  MoveL (T10079) to (119.5, 116.18, 12.1) mm, rotated rx 180 ry 0 rz -180 deg; joints [0, 0, 0, 0, 0, 0]
  Call Extruder -0.04075
  MoveL (T10080) to (119.58, 116.26, 12.1) mm, rotated rx 180 ry 0 rz -180 deg; joints [0, 0, 0, 0, 0, 0]
  Call Extruder -0.07305
  MoveL (T10081) to (119.79, 116.26, 12.1) mm, rotated rx 180 ry 0 rz -180 deg; joints [0, 0, 0, 0, 0, 0]
  Call Extruder -0.05902
  MoveL (T10082) to (119.9, 116.14, 12.1) mm, rotated rx 180 ry 0 rz -180 deg; joints [0, 0, 0, 0, 0, 0]
  Set speed (45.0 mm/s)
  Call Extruder -0.02
  MoveL (T10083) to (119.9, 116.14, 12.1) mm, rotated rx 180 ry 0 rz -180 deg; joints [0, 0, 0, 0, 0, 0]
  Set speed (150.0 mm/s)
  MoveL (T10084) to (119.9, 116.14, 14.1) mm, rotated rx 180 ry 0 rz -180 deg; joints [0, 0, 0, 0, 0, 0]
  MoveL (T10085) to (104.34, 103.54, 14.1) mm, rotated rx 180 ry 0 rz -180 deg; joints [0, 0, 0, 0, 0, 0]
  MoveL (T10086) to (104.34, 103.54, 12.3) mm, rotated rx 180 ry 0 rz -180 deg; joints [0, 0, 0, 0, 0, 0]
  Set speed (40.0 mm/s)
  Call Extruder 2.0
  MoveL (T10087) to (104.34, 103.54, 12.3) mm, rotated rx 180 ry 0 rz -180 deg; joints [0, 0, 0, 0, 0, 0]
  Set speed (26.4 mm/s)
  MoveL (T10088) to (104.34, 103.54, 12.3) mm, rotated rx 180 ry 0 rz -180 deg; joints [0, 0, 0, 0, 0, 0]
  Call Extruder 0.13732
  MoveL (T10089) to (108.85, 103.54, 12.3) mm, rotated rx 180 ry 0 rz -180 deg; joints [0, 0, 0, 0, 0, 0]
  Call Extruder 0.05783
  MoveL (T10090) to (108.85, 105.44, 12.3) mm, rotated rx 180 ry 0 rz -180 deg; joints [0, 0, 0, 0, 0, 0]
  Call Extruder 0.1948
  MoveL (T10091) to (115.24, 105.44, 12.3) mm, rotated rx 180 ry 0 rz -180 deg; joints [0, 0, 0, 0, 0, 0]
  Call Extruder 0.05783
  MoveL (T10092) to (115.24, 103.54, 12.3) mm, rotated rx 180 ry 0 rz -180 deg; joints [0, 0, 0, 0, 0, 0]
  Call Extruder 0.18953
  MoveL (T10093) to (121.46, 103.54, 12.3) mm, rotated rx 180 ry 0 rz -180 deg; joints [0, 0, 0, 0, 0, 0]
  Call Extruder 0.14944
  MoveL (T10094) to (121.46, 108.44, 12.3) mm, rotated rx 180 ry 0 rz -180 deg; joints [0, 0, 0, 0, 0, 0]
  Call Extruder 0.05883
  MoveL (T10095) to (119.53, 108.44, 12.3) mm, rotated rx 180 ry 0 rz -180 deg; joints [0, 0, 0, 0, 0, 0]
  Call Extruder 0.22006
  MoveL (T10096) to (119.53, 115.67, 12.3) mm, rotated rx 180 ry 0 rz -180 deg; joints [0, 0, 0, 0, 0, 0]
  Call Extruder 0.05893
  MoveL (T10097) to (121.46, 115.67, 12.3) mm, rotated rx 180 ry 0 rz -180 deg; joints [0, 0, 0, 0, 0, 0]
  Call Extruder 0.17636
  MoveL (T10098) to (121.46, 121.46, 12.3) mm, rotated rx 180 ry 0 rz -180 deg; joints [0, 0, 0, 0, 0, 0]
  Call Extruder 0.54596
  MoveL (T10099) to (103.54, 121.46, 12.3) mm, rotated rx 180 ry 0 rz -180 deg; joints [0, 0, 0, 0, 0, 0]
  Call Extruder 0.54596
  MoveL (T10100) to (103.54, 103.54, 12.3) mm, rotated rx 180 ry 0 rz -180 deg; joints [0, 0, 0, 0, 0, 0]
  Call Extruder 0.02254
  MoveL (T10101) to (104.28, 103.54, 12.3) mm, rotated rx 180 ry 0 rz -180 deg; joints [0, 0, 0, 0, 0, 0]
  Set speed (150.0 mm/s)
  MoveL (T10102) to (103.53, 103.13, 12.3) mm, rotated rx 180 ry 0 rz -180 deg; joints [0, 0, 0, 0, 0, 0]
  Set speed (26.4 mm/s)
  MoveL (T10103) to (103.53, 103.13, 12.3) mm, rotated rx 180 ry 0 rz -180 deg; joints [0, 0, 0, 0, 0, 0]
  Call Extruder 0.17431
  MoveL (T10104) to (109.25, 103.13, 12.3) mm, rotated rx 180 ry 0 rz -180 deg; joints [0, 0, 0, 0, 0, 0]
  Call Extruder 0.05783
  MoveL (T10105) to (109.25, 105.03, 12.3) mm, rotated rx 180 ry 0 rz -180 deg; joints [0, 0, 0, 0, 0, 0]
  Call Extruder 0.08214
  MoveL (T10106) to (111.95, 105.03, 12.3) mm, rotated rx 180 ry 0 rz -180 deg; joints [0, 0, 0, 0, 0, 0]
  Call Extruder 0.08784
  MoveL (T10107) to (114.83, 105.03, 12.3) mm, rotated rx 180 ry 0 rz -180 deg; joints [0, 0, 0, 0, 0, 0]
  Call Extruder 0.05783
  MoveL (T10108) to (114.83, 103.13, 12.3) mm, rotated rx 180 ry 0 rz -180 deg; joints [0, 0, 0, 0, 0, 0]
  Call Extruder 0.21434
  MoveL (T10109) to (121.87, 103.13, 12.3) mm, rotated rx 180 ry 0 rz -180 deg; joints [0, 0, 0, 0, 0, 0]
  Call Extruder 0.17423
  MoveL (T10110) to (121.87, 108.85, 12.3) mm, rotated rx 180 ry 0 rz -180 deg; joints [0, 0, 0, 0, 0, 0]
  Call Extruder 0.05884
  MoveL (T10111) to (119.94, 108.85, 12.3) mm, rotated rx 180 ry 0 rz -180 deg; joints [0, 0, 0, 0, 0, 0]
  Call Extruder 0.09005
  MoveL (T10112) to (119.94, 111.81, 12.3) mm, rotated rx 180 ry 0 rz -180 deg; joints [0, 0, 0, 0, 0, 0]
  Call Extruder 0.05887
  MoveL (T10113) to (121.87, 111.81, 12.3) mm, rotated rx 180 ry 0 rz -180 deg; joints [0, 0, 0, 0, 0, 0]
  Call Extruder 0.01564
  MoveL (T10114) to (121.87, 112.32, 12.3) mm, rotated rx 180 ry 0 rz -180 deg; joints [0, 0, 0, 0, 0, 0]
  Call Extruder 0.05888
  MoveL (T10115) to (119.94, 112.32, 12.3) mm, rotated rx 180 ry 0 rz -180 deg; joints [0, 0, 0, 0, 0, 0]
  Call Extruder 0.08969
  MoveL (T10116) to (119.93, 115.26, 12.3) mm, rotated rx 180 ry 0 rz -180 deg; joints [0, 0, 0, 0, 0, 0]
  Call Extruder 0.05892
  MoveL (T10117) to (121.87, 115.27, 12.3) mm, rotated rx 180 ry 0 rz -180 deg; joints [0, 0, 0, 0, 0, 0]
  Call Extruder 0.20115
  MoveL (T10118) to (121.87, 121.87, 12.3) mm, rotated rx 180 ry 0 rz -180 deg; joints [0, 0, 0, 0, 0, 0]
  Call Extruder 0.57077
  MoveL (T10119) to (103.13, 121.87, 12.3) mm, rotated rx 180 ry 0 rz -180 deg; joints [0, 0, 0, 0, 0, 0]
  Call Extruder 0.57077
  MoveL (T10120) to (103.13, 103.13, 12.3) mm, rotated rx 180 ry 0 rz -180 deg; joints [0, 0, 0, 0, 0, 0]
  Call Extruder 0.01036
  MoveL (T10121) to (103.47, 103.13, 12.3) mm, rotated rx 180 ry 0 rz -180 deg; joints [0, 0, 0, 0, 0, 0]
  Set speed (150.0 mm/s)
  MoveL (T10122) to (102.72, 102.81, 12.3) mm, rotated rx 180 ry 0 rz -180 deg; joints [0, 0, 0, 0, 0, 0]
  Set speed (25.0 mm/s)
  MoveL (T10123) to (102.72, 102.81, 12.3) mm, rotated rx 180 ry 0 rz -180 deg; joints [0, 0, 0, 0, 0, 0]
  Call Extruder 0.00259
  MoveL (T10124) to (102.72, 102.72, 12.3) mm, rotated rx 180 ry 0 rz -180 deg; joints [0, 0, 0, 0, 0, 0]
  Call Extruder 0.21131
  MoveL (T10125) to (109.66, 102.72, 12.3) mm, rotated rx 180 ry 0 rz -180 deg; joints [0, 0, 0, 0, 0, 0]
  Call Extruder 0.05783
  MoveL (T10126) to (109.66, 104.62, 12.3) mm, rotated rx 180 ry 0 rz -180 deg; joints [0, 0, 0, 0, 0, 0]
  Call Extruder 0.0643
  MoveL (T10127) to (111.77, 104.62, 12.3) mm, rotated rx 180 ry 0 rz -180 deg; joints [0, 0, 0, 0, 0, 0]
  Call Extruder 0.05783
  MoveL (T10128) to (111.77, 102.72, 12.3) mm, rotated rx 180 ry 0 rz -180 deg; joints [0, 0, 0, 0, 0, 0]
  Call Extruder 0.01777
  MoveL (T10129) to (112.36, 102.72, 12.3) mm, rotated rx 180 ry 0 rz -180 deg; joints [0, 0, 0, 0, 0, 0]
  Call Extruder 0.05783
  MoveL (T10130) to (112.36, 104.62, 12.3) mm, rotated rx 180 ry 0 rz -180 deg; joints [0, 0, 0, 0, 0, 0]
  Call Extruder 0.06304
  MoveL (T10131) to (114.43, 104.62, 12.3) mm, rotated rx 180 ry 0 rz -180 deg; joints [0, 0, 0, 0, 0, 0]
  Call Extruder 0.05783
  MoveL (T10132) to (114.42, 102.72, 12.3) mm, rotated rx 180 ry 0 rz -180 deg; joints [0, 0, 0, 0, 0, 0]
  Call Extruder 0.23915
  MoveL (T10133) to (122.28, 102.72, 12.3) mm, rotated rx 180 ry 0 rz -180 deg; joints [0, 0, 0, 0, 0, 0]
  Call Extruder 0.19903
  MoveL (T10134) to (122.28, 109.26, 12.3) mm, rotated rx 180 ry 0 rz -180 deg; joints [0, 0, 0, 0, 0, 0]
  Call Extruder 0.05884
  MoveL (T10135) to (120.34, 109.26, 12.3) mm, rotated rx 180 ry 0 rz -180 deg; joints [0, 0, 0, 0, 0, 0]
  Call Extruder 0.06525
  MoveL (T10136) to (120.34, 111.4, 12.3) mm, rotated rx 180 ry 0 rz -180 deg; joints [0, 0, 0, 0, 0, 0]
  Call Extruder 0.05887
  MoveL (T10137) to (122.28, 111.4, 12.3) mm, rotated rx 180 ry 0 rz -180 deg; joints [0, 0, 0, 0, 0, 0]
  Call Extruder 0.04047
  MoveL (T10138) to (122.28, 112.73, 12.3) mm, rotated rx 180 ry 0 rz -180 deg; joints [0, 0, 0, 0, 0, 0]
  Call Extruder 0.05889
  MoveL (T10139) to (120.34, 112.73, 12.3) mm, rotated rx 180 ry 0 rz -180 deg; joints [0, 0, 0, 0, 0, 0]
  Call Extruder 0.06488
  MoveL (T10140) to (120.34, 114.86, 12.3) mm, rotated rx 180 ry 0 rz -180 deg; joints [0, 0, 0, 0, 0, 0]
  Call Extruder 0.05892
  MoveL (T10141) to (122.28, 114.86, 12.3) mm, rotated rx 180 ry 0 rz -180 deg; joints [0, 0, 0, 0, 0, 0]
  Call Extruder 0.22594
  MoveL (T10142) to (122.28, 122.28, 12.3) mm, rotated rx 180 ry 0 rz -180 deg; joints [0, 0, 0, 0, 0, 0]
  Call Extruder 0.59557
  MoveL (T10143) to (102.72, 122.28, 12.3) mm, rotated rx 180 ry 0 rz -180 deg; joints [0, 0, 0, 0, 0, 0]
  Call Extruder 0.59115
  MoveL (T10144) to (102.72, 102.87, 12.3) mm, rotated rx 180 ry 0 rz -180 deg; joints [0, 0, 0, 0, 0, 0]
  Set speed (150.0 mm/s)
  MoveL (T10145) to (102.78, 102.75, 12.3) mm, rotated rx 180 ry 0 rz -180 deg; joints [0, 0, 0, 0, 0, 0]
  Set speed (45.0 mm/s)
  Call Extruder -1.6
  MoveL (T10146) to (102.78, 102.75, 12.3) mm, rotated rx 180 ry 0 rz -180 deg; joints [0, 0, 0, 0, 0, 0]
  Set speed (120.0 mm/s)
  MoveL (T10147) to (102.78, 102.75, 12.3) mm, rotated rx 180 ry 0 rz -180 deg; joints [0, 0, 0, 0, 0, 0]
  Call Extruder -0.05166
  MoveL (T10148) to (102.72, 102.72, 12.3) mm, rotated rx 180 ry 0 rz -180 deg; joints [0, 0, 0, 0, 0, 0]
  Call Extruder -0.32834
  MoveL (T10149) to (103.65, 102.72, 12.3) mm, rotated rx 180 ry 0 rz -180 deg; joints [0, 0, 0, 0, 0, 0]
  Set speed (45.0 mm/s)
  Call Extruder -0.02
  MoveL (T10150) to (103.65, 102.72, 12.3) mm, rotated rx 180 ry 0 rz -180 deg; joints [0, 0, 0, 0, 0, 0]
  Set speed (150.0 mm/s)
  MoveL (T10151) to (103.65, 102.72, 14.3) mm, rotated rx 180 ry 0 rz -180 deg; joints [0, 0, 0, 0, 0, 0]
  MoveL (T10152) to (106.29, 103.84, 14.3) mm, rotated rx 180 ry 0 rz -180 deg; joints [0, 0, 0, 0, 0, 0]
  MoveL (T10153) to (106.29, 103.84, 12.3) mm, rotated rx 180 ry 0 rz -180 deg; joints [0, 0, 0, 0, 0, 0]
  Set speed (40.0 mm/s)
  Call Extruder 2.0
  MoveL (T10154) to (106.29, 103.84, 12.3) mm, rotated rx 180 ry 0 rz -180 deg; joints [0, 0, 0, 0, 0, 0]
  Set speed (26.4 mm/s)
  MoveL (T10155) to (106.29, 103.84, 12.3) mm, rotated rx 180 ry 0 rz -180 deg; joints [0, 0, 0, 0, 0, 0]
  Call Extruder 0.07441
  MoveL (T10156) to (103.84, 103.84, 12.3) mm, rotated rx 180 ry 0 rz -180 deg; joints [0, 0, 0, 0, 0, 0]
  Call Extruder 0.7458
  MoveL (T10157) to (121.16, 121.16, 12.3) mm, rotated rx 180 ry 0 rz -180 deg; joints [0, 0, 0, 0, 0, 0]
  Call Extruder 0.10645
  MoveL (T10158) to (121.16, 117.66, 12.3) mm, rotated rx 180 ry 0 rz -180 deg; joints [0, 0, 0, 0, 0, 0]
  Call Extruder 0.15054
  MoveL (T10159) to (117.66, 121.16, 12.3) mm, rotated rx 180 ry 0 rz -180 deg; joints [0, 0, 0, 0, 0, 0]
  Call Extruder 0.03385
  MoveL (T10160) to (116.55, 121.16, 12.3) mm, rotated rx 180 ry 0 rz -180 deg; joints [0, 0, 0, 0, 0, 0]
  Call Extruder 0.54738
  MoveL (T10161) to (103.84, 108.45, 12.3) mm, rotated rx 180 ry 0 rz -180 deg; joints [0, 0, 0, 0, 0, 0]
  Call Extruder 0.03385
  MoveL (T10162) to (103.84, 107.34, 12.3) mm, rotated rx 180 ry 0 rz -180 deg; joints [0, 0, 0, 0, 0, 0]
  Call Extruder 0.15054
  MoveL (T10163) to (107.34, 103.84, 12.3) mm, rotated rx 180 ry 0 rz -180 deg; joints [0, 0, 0, 0, 0, 0]
  Call Extruder 0.01217
  MoveL (T10164) to (107.74, 103.84, 12.3) mm, rotated rx 180 ry 0 rz -180 deg; joints [0, 0, 0, 0, 0, 0]
  Call Extruder 0.05203
  MoveL (T10165) to (107.74, 105.55, 12.3) mm, rotated rx 180 ry 0 rz -180 deg; joints [0, 0, 0, 0, 0, 0]
  Call Extruder 0.01021
  MoveL (T10166) to (107.97, 105.79, 12.3) mm, rotated rx 180 ry 0 rz -180 deg; joints [0, 0, 0, 0, 0, 0]
  Set speed (150.0 mm/s)
  MoveL (T10167) to (107.96, 103.84, 12.3) mm, rotated rx 180 ry 0 rz -180 deg; joints [0, 0, 0, 0, 0, 0]
  Set speed (26.4 mm/s)
  MoveL (T10168) to (107.96, 103.84, 12.3) mm, rotated rx 180 ry 0 rz -180 deg; joints [0, 0, 0, 0, 0, 0]
  Call Extruder 0.0285
  MoveL (T10169) to (108.54, 104.42, 12.3) mm, rotated rx 180 ry 0 rz -180 deg; joints [0, 0, 0, 0, 0, 0]
  Call Extruder 0.02289
  MoveL (T10170) to (108.54, 105.08, 12.3) mm, rotated rx 180 ry 0 rz -180 deg; joints [0, 0, 0, 0, 0, 0]
  Call Extruder 0.01948
  MoveL (T10171) to (108.14, 104.69, 12.3) mm, rotated rx 180 ry 0 rz -180 deg; joints [0, 0, 0, 0, 0, 0]
  Call Extruder 0.02289
  MoveL (T10172) to (108.14, 105.34, 12.3) mm, rotated rx 180 ry 0 rz -180 deg; joints [0, 0, 0, 0, 0, 0]
  Call Extruder 0.01503
  MoveL (T10173) to (108.45, 105.65, 12.3) mm, rotated rx 180 ry 0 rz -180 deg; joints [0, 0, 0, 0, 0, 0]
  Set speed (45.0 mm/s)
  Call Extruder -1.6
  MoveL (T10174) to (108.45, 105.65, 12.3) mm, rotated rx 180 ry 0 rz -180 deg; joints [0, 0, 0, 0, 0, 0]
  Set speed (120.0 mm/s)
  MoveL (T10175) to (108.45, 105.65, 12.3) mm, rotated rx 180 ry 0 rz -180 deg; joints [0, 0, 0, 0, 0, 0]
  Call Extruder -0.15377
  MoveL (T10176) to (108.14, 105.34, 12.3) mm, rotated rx 180 ry 0 rz -180 deg; joints [0, 0, 0, 0, 0, 0]
  Call Extruder -0.22623
  MoveL (T10177) to (108.14, 104.71, 12.3) mm, rotated rx 180 ry 0 rz -180 deg; joints [0, 0, 0, 0, 0, 0]
  Set speed (45.0 mm/s)
  Call Extruder -0.02
  MoveL (T10178) to (108.14, 104.71, 12.3) mm, rotated rx 180 ry 0 rz -180 deg; joints [0, 0, 0, 0, 0, 0]
  Set speed (150.0 mm/s)
  MoveL (T10179) to (108.14, 104.71, 14.3) mm, rotated rx 180 ry 0 rz -180 deg; joints [0, 0, 0, 0, 0, 0]
  MoveL (T10180) to (112.06, 104.83, 14.3) mm, rotated rx 180 ry 0 rz -180 deg; joints [0, 0, 0, 0, 0, 0]
  MoveL (T10181) to (112.06, 104.83, 12.3) mm, rotated rx 180 ry 0 rz -180 deg; joints [0, 0, 0, 0, 0, 0]
  Set speed (40.0 mm/s)
  Call Extruder 2.0
  MoveL (T10182) to (112.06, 104.83, 12.3) mm, rotated rx 180 ry 0 rz -180 deg; joints [0, 0, 0, 0, 0, 0]
  Set speed (26.4 mm/s)
  MoveL (T10183) to (112.06, 104.83, 12.3) mm, rotated rx 180 ry 0 rz -180 deg; joints [0, 0, 0, 0, 0, 0]
  Call Extruder 0.02531
  MoveL (T10184) to (112.06, 102.93, 12.3) mm, rotated rx 180 ry 0 rz -180 deg; joints [0, 0, 0, 0, 0, 0]
  Set speed (45.0 mm/s)
  Call Extruder -1.6
  MoveL (T10185) to (112.06, 102.93, 12.3) mm, rotated rx 180 ry 0 rz -180 deg; joints [0, 0, 0, 0, 0, 0]
  Set speed (120.0 mm/s)
  MoveL (T10186) to (112.06, 102.93, 12.3) mm, rotated rx 180 ry 0 rz -180 deg; joints [0, 0, 0, 0, 0, 0]
  Call Extruder -0.38
  MoveL (T10187) to (112.06, 104, 12.3) mm, rotated rx 180 ry 0 rz -180 deg; joints [0, 0, 0, 0, 0, 0]
  Set speed (45.0 mm/s)
  Call Extruder -0.02
  MoveL (T10188) to (112.06, 104, 12.3) mm, rotated rx 180 ry 0 rz -180 deg; joints [0, 0, 0, 0, 0, 0]
  Set speed (150.0 mm/s)
  MoveL (T10189) to (112.06, 104, 14.3) mm, rotated rx 180 ry 0 rz -180 deg; joints [0, 0, 0, 0, 0, 0]
  MoveL (T10190) to (115.84, 103.66, 14.3) mm, rotated rx 180 ry 0 rz -180 deg; joints [0, 0, 0, 0, 0, 0]
  MoveL (T10191) to (115.84, 103.66, 12.3) mm, rotated rx 180 ry 0 rz -180 deg; joints [0, 0, 0, 0, 0, 0]
  Set speed (40.0 mm/s)
  Call Extruder 2.0
  MoveL (T10192) to (115.84, 103.66, 12.3) mm, rotated rx 180 ry 0 rz -180 deg; joints [0, 0, 0, 0, 0, 0]
  Set speed (26.4 mm/s)
  MoveL (T10193) to (115.84, 103.66, 12.3) mm, rotated rx 180 ry 0 rz -180 deg; joints [0, 0, 0, 0, 0, 0]
  Call Extruder 0.01001
  MoveL (T10194) to (116.03, 103.86, 12.3) mm, rotated rx 180 ry 0 rz -180 deg; joints [0, 0, 0, 0, 0, 0]
  Call Extruder 0.02527
  MoveL (T10195) to (116.03, 104.55, 12.3) mm, rotated rx 180 ry 0 rz -180 deg; joints [0, 0, 0, 0, 0, 0]
  Call Extruder 0.02525
  MoveL (T10196) to (115.55, 104.06, 12.3) mm, rotated rx 180 ry 0 rz -180 deg; joints [0, 0, 0, 0, 0, 0]
  Call Extruder 0.02527
  MoveL (T10197) to (115.55, 104.75, 12.3) mm, rotated rx 180 ry 0 rz -180 deg; joints [0, 0, 0, 0, 0, 0]
  Call Extruder 0.02525
  MoveL (T10198) to (116.03, 105.24, 12.3) mm, rotated rx 180 ry 0 rz -180 deg; joints [0, 0, 0, 0, 0, 0]
  Call Extruder 0.00536
  MoveL (T10199) to (116.03, 105.38, 12.3) mm, rotated rx 180 ry 0 rz -180 deg; joints [0, 0, 0, 0, 0, 0]
  Call Extruder 0.00419
  MoveL (T10200) to (115.95, 105.47, 12.3) mm, rotated rx 180 ry 0 rz -180 deg; joints [0, 0, 0, 0, 0, 0]
  Call Extruder 0.01397
  MoveL (T10201) to (115.57, 105.47, 12.3) mm, rotated rx 180 ry 0 rz -180 deg; joints [0, 0, 0, 0, 0, 0]
  Call Extruder 0.01077
  MoveL (T10202) to (115.36, 105.26, 12.3) mm, rotated rx 180 ry 0 rz -180 deg; joints [0, 0, 0, 0, 0, 0]
  Set speed (150.0 mm/s)
  MoveL (T10203) to (115.73, 105.87, 12.3) mm, rotated rx 180 ry 0 rz -180 deg; joints [0, 0, 0, 0, 0, 0]
  Set speed (26.4 mm/s)
  MoveL (T10204) to (115.73, 105.87, 12.3) mm, rotated rx 180 ry 0 rz -180 deg; joints [0, 0, 0, 0, 0, 0]
  Call Extruder 0.01195
  MoveL (T10205) to (116.12, 105.87, 12.3) mm, rotated rx 180 ry 0 rz -180 deg; joints [0, 0, 0, 0, 0, 0]
  Call Extruder 0.01377
  MoveL (T10206) to (116.44, 105.55, 12.3) mm, rotated rx 180 ry 0 rz -180 deg; joints [0, 0, 0, 0, 0, 0]
  Call Extruder 0.04869
  MoveL (T10207) to (116.44, 103.95, 12.3) mm, rotated rx 180 ry 0 rz -180 deg; joints [0, 0, 0, 0, 0, 0]
  Call Extruder 0.00473
  MoveL (T10208) to (116.55, 103.84, 12.3) mm, rotated rx 180 ry 0 rz -180 deg; joints [0, 0, 0, 0, 0, 0]
  Call Extruder 0.03385
  MoveL (T10209) to (117.66, 103.84, 12.3) mm, rotated rx 180 ry 0 rz -180 deg; joints [0, 0, 0, 0, 0, 0]
  Call Extruder 0.14859
  MoveL (T10210) to (121.11, 107.29, 12.3) mm, rotated rx 180 ry 0 rz -180 deg; joints [0, 0, 0, 0, 0, 0]
  Call Extruder 0.00138
  MoveL (T10211) to (121.16, 107.29, 12.3) mm, rotated rx 180 ry 0 rz -180 deg; joints [0, 0, 0, 0, 0, 0]
  Call Extruder 0.10507
  MoveL (T10212) to (121.16, 103.84, 12.3) mm, rotated rx 180 ry 0 rz -180 deg; joints [0, 0, 0, 0, 0, 0]
  Call Extruder 0.7458
  MoveL (T10213) to (103.84, 121.16, 12.3) mm, rotated rx 180 ry 0 rz -180 deg; joints [0, 0, 0, 0, 0, 0]
  Call Extruder 0.10645
  MoveL (T10214) to (103.84, 117.66, 12.3) mm, rotated rx 180 ry 0 rz -180 deg; joints [0, 0, 0, 0, 0, 0]
  Call Extruder 0.15054
  MoveL (T10215) to (107.34, 121.16, 12.3) mm, rotated rx 180 ry 0 rz -180 deg; joints [0, 0, 0, 0, 0, 0]
  Call Extruder 0.03385
  MoveL (T10216) to (108.45, 121.16, 12.3) mm, rotated rx 180 ry 0 rz -180 deg; joints [0, 0, 0, 0, 0, 0]
  Call Extruder 0.46415
  MoveL (T10217) to (119.22, 110.38, 12.3) mm, rotated rx 180 ry 0 rz -180 deg; joints [0, 0, 0, 0, 0, 0]
  Call Extruder 0.01126
  MoveL (T10218) to (119.22, 110.01, 12.3) mm, rotated rx 180 ry 0 rz -180 deg; joints [0, 0, 0, 0, 0, 0]
  Call Extruder 0.18395
  MoveL (T10219) to (114.95, 105.74, 12.3) mm, rotated rx 180 ry 0 rz -180 deg; joints [0, 0, 0, 0, 0, 0]
  Call Extruder 0.00922
  MoveL (T10220) to (114.65, 105.74, 12.3) mm, rotated rx 180 ry 0 rz -180 deg; joints [0, 0, 0, 0, 0, 0]
  Call Extruder 0.46559
  MoveL (T10221) to (103.84, 116.55, 12.3) mm, rotated rx 180 ry 0 rz -180 deg; joints [0, 0, 0, 0, 0, 0]
  Call Extruder 0.10645
  MoveL (T10222) to (103.84, 113.06, 12.3) mm, rotated rx 180 ry 0 rz -180 deg; joints [0, 0, 0, 0, 0, 0]
  Call Extruder 0.34896
  MoveL (T10223) to (111.94, 121.16, 12.3) mm, rotated rx 180 ry 0 rz -180 deg; joints [0, 0, 0, 0, 0, 0]
  Call Extruder 0.03385
  MoveL (T10224) to (113.06, 121.16, 12.3) mm, rotated rx 180 ry 0 rz -180 deg; joints [0, 0, 0, 0, 0, 0]
  Call Extruder 0.26564
  MoveL (T10225) to (119.22, 114.99, 12.3) mm, rotated rx 180 ry 0 rz -180 deg; joints [0, 0, 0, 0, 0, 0]
  Call Extruder 0.01138
  MoveL (T10226) to (119.22, 114.62, 12.3) mm, rotated rx 180 ry 0 rz -180 deg; joints [0, 0, 0, 0, 0, 0]
  Call Extruder 0.38228
  MoveL (T10227) to (110.35, 105.74, 12.3) mm, rotated rx 180 ry 0 rz -180 deg; joints [0, 0, 0, 0, 0, 0]
  Call Extruder 0.00922
  MoveL (T10228) to (110.05, 105.74, 12.3) mm, rotated rx 180 ry 0 rz -180 deg; joints [0, 0, 0, 0, 0, 0]
  Call Extruder 0.26717
  MoveL (T10229) to (103.84, 111.94, 12.3) mm, rotated rx 180 ry 0 rz -180 deg; joints [0, 0, 0, 0, 0, 0]
  Call Extruder 0.07441
  MoveL (T10230) to (103.84, 109.5, 12.3) mm, rotated rx 180 ry 0 rz -180 deg; joints [0, 0, 0, 0, 0, 0]
  Set speed (45.0 mm/s)
  Call Extruder -1.6
  MoveL (T10231) to (103.84, 109.5, 12.3) mm, rotated rx 180 ry 0 rz -180 deg; joints [0, 0, 0, 0, 0, 0]
  Set speed (120.0 mm/s)
  MoveL (T10232) to (103.84, 109.5, 12.3) mm, rotated rx 180 ry 0 rz -180 deg; joints [0, 0, 0, 0, 0, 0]
  Call Extruder -0.38
  MoveL (T10233) to (103.84, 110.57, 12.3) mm, rotated rx 180 ry 0 rz -180 deg; joints [0, 0, 0, 0, 0, 0]
  Set speed (45.0 mm/s)
  Call Extruder -0.02
  MoveL (T10234) to (103.84, 110.57, 12.3) mm, rotated rx 180 ry 0 rz -180 deg; joints [0, 0, 0, 0, 0, 0]
  Set speed (150.0 mm/s)
  MoveL (T10235) to (103.84, 110.57, 14.3) mm, rotated rx 180 ry 0 rz -180 deg; joints [0, 0, 0, 0, 0, 0]
  MoveL (T10236) to (119.73, 112.06, 14.3) mm, rotated rx 180 ry 0 rz -180 deg; joints [0, 0, 0, 0, 0, 0]
  MoveL (T10237) to (119.73, 112.06, 12.3) mm, rotated rx 180 ry 0 rz -180 deg; joints [0, 0, 0, 0, 0, 0]
  Set speed (40.0 mm/s)
  Call Extruder 2.0
  MoveL (T10238) to (119.73, 112.06, 12.3) mm, rotated rx 180 ry 0 rz -180 deg; joints [0, 0, 0, 0, 0, 0]
  Set speed (26.4 mm/s)
  MoveL (T10239) to (119.73, 112.06, 12.3) mm, rotated rx 180 ry 0 rz -180 deg; joints [0, 0, 0, 0, 0, 0]
  Call Extruder 0.01533
  MoveL (T10240) to (121.66, 112.06, 12.3) mm, rotated rx 180 ry 0 rz -180 deg; joints [0, 0, 0, 0, 0, 0]
  Set speed (45.0 mm/s)
  Call Extruder -1.6
  MoveL (T10241) to (121.66, 112.06, 12.3) mm, rotated rx 180 ry 0 rz -180 deg; joints [0, 0, 0, 0, 0, 0]
  Set speed (120.0 mm/s)
  MoveL (T10242) to (121.66, 112.06, 12.3) mm, rotated rx 180 ry 0 rz -180 deg; joints [0, 0, 0, 0, 0, 0]
  Call Extruder -0.38
  MoveL (T10243) to (120.6, 112.06, 12.3) mm, rotated rx 180 ry 0 rz -180 deg; joints [0, 0, 0, 0, 0, 0]
  Set speed (45.0 mm/s)
  Call Extruder -0.02
  MoveL (T10244) to (120.6, 112.06, 12.3) mm, rotated rx 180 ry 0 rz -180 deg; joints [0, 0, 0, 0, 0, 0]
  Set speed (150.0 mm/s)
  MoveL (T10245) to (120.6, 112.06, 14.3) mm, rotated rx 180 ry 0 rz -180 deg; joints [0, 0, 0, 0, 0, 0]
  MoveL (T10246) to (121.34, 107.89, 14.3) mm, rotated rx 180 ry 0 rz -180 deg; joints [0, 0, 0, 0, 0, 0]
  MoveL (T10247) to (121.34, 107.89, 12.3) mm, rotated rx 180 ry 0 rz -180 deg; joints [0, 0, 0, 0, 0, 0]
  Set speed (40.0 mm/s)
  Call Extruder 2.0
  MoveL (T10248) to (121.34, 107.89, 12.3) mm, rotated rx 180 ry 0 rz -180 deg; joints [0, 0, 0, 0, 0, 0]
  Set speed (26.4 mm/s)
  MoveL (T10249) to (121.34, 107.89, 12.3) mm, rotated rx 180 ry 0 rz -180 deg; joints [0, 0, 0, 0, 0, 0]
  Call Extruder 0.00999
  MoveL (T10250) to (121.14, 107.7, 12.3) mm, rotated rx 180 ry 0 rz -180 deg; joints [0, 0, 0, 0, 0, 0]
  Call Extruder 0.0252
  MoveL (T10251) to (120.45, 107.7, 12.3) mm, rotated rx 180 ry 0 rz -180 deg; joints [0, 0, 0, 0, 0, 0]
  Call Extruder 0.02266
  MoveL (T10252) to (120.89, 108.14, 12.3) mm, rotated rx 180 ry 0 rz -180 deg; joints [0, 0, 0, 0, 0, 0]
  Call Extruder 0.0252
  MoveL (T10253) to (120.2, 108.14, 12.3) mm, rotated rx 180 ry 0 rz -180 deg; joints [0, 0, 0, 0, 0, 0]
  Call Extruder 0.02266
  MoveL (T10254) to (119.77, 107.7, 12.3) mm, rotated rx 180 ry 0 rz -180 deg; joints [0, 0, 0, 0, 0, 0]
  Call Extruder 0.00655
  MoveL (T10255) to (119.59, 107.7, 12.3) mm, rotated rx 180 ry 0 rz -180 deg; joints [0, 0, 0, 0, 0, 0]
  Call Extruder 0.00418
  MoveL (T10256) to (119.5, 107.78, 12.3) mm, rotated rx 180 ry 0 rz -180 deg; joints [0, 0, 0, 0, 0, 0]
  Call Extruder 0.01271
  MoveL (T10257) to (119.5, 108.13, 12.3) mm, rotated rx 180 ry 0 rz -180 deg; joints [0, 0, 0, 0, 0, 0]
  Call Extruder 0.00998
  MoveL (T10258) to (119.7, 108.32, 12.3) mm, rotated rx 180 ry 0 rz -180 deg; joints [0, 0, 0, 0, 0, 0]
  Set speed (45.0 mm/s)
  Call Extruder -1.6
  MoveL (T10259) to (119.7, 108.32, 12.3) mm, rotated rx 180 ry 0 rz -180 deg; joints [0, 0, 0, 0, 0, 0]
  Set speed (120.0 mm/s)
  MoveL (T10260) to (119.7, 108.32, 12.3) mm, rotated rx 180 ry 0 rz -180 deg; joints [0, 0, 0, 0, 0, 0]
  Call Extruder -0.09732
  MoveL (T10261) to (119.5, 108.13, 12.3) mm, rotated rx 180 ry 0 rz -180 deg; joints [0, 0, 0, 0, 0, 0]
  Call Extruder -0.12397
  MoveL (T10262) to (119.5, 107.78, 12.3) mm, rotated rx 180 ry 0 rz -180 deg; joints [0, 0, 0, 0, 0, 0]
  Call Extruder -0.04075
  MoveL (T10263) to (119.59, 107.7, 12.3) mm, rotated rx 180 ry 0 rz -180 deg; joints [0, 0, 0, 0, 0, 0]
  Call Extruder -0.06391
  MoveL (T10264) to (119.77, 107.7, 12.3) mm, rotated rx 180 ry 0 rz -180 deg; joints [0, 0, 0, 0, 0, 0]
  Call Extruder -0.05404
  MoveL (T10265) to (119.87, 107.81, 12.3) mm, rotated rx 180 ry 0 rz -180 deg; joints [0, 0, 0, 0, 0, 0]
  Set speed (45.0 mm/s)
  Call Extruder -0.02
  MoveL (T10266) to (119.87, 107.81, 12.3) mm, rotated rx 180 ry 0 rz -180 deg; joints [0, 0, 0, 0, 0, 0]
  Set speed (150.0 mm/s)
  MoveL (T10267) to (119.87, 107.81, 14.3) mm, rotated rx 180 ry 0 rz -180 deg; joints [0, 0, 0, 0, 0, 0]
  MoveL (T10268) to (121.15, 116.56, 14.3) mm, rotated rx 180 ry 0 rz -180 deg; joints [0, 0, 0, 0, 0, 0]
  MoveL (T10269) to (121.15, 116.56, 12.3) mm, rotated rx 180 ry 0 rz -180 deg; joints [0, 0, 0, 0, 0, 0]
  Set speed (40.0 mm/s)
  Call Extruder 2.0
  MoveL (T10270) to (121.15, 116.56, 12.3) mm, rotated rx 180 ry 0 rz -180 deg; joints [0, 0, 0, 0, 0, 0]
  Set speed (26.4 mm/s)
  MoveL (T10271) to (121.15, 116.56, 12.3) mm, rotated rx 180 ry 0 rz -180 deg; joints [0, 0, 0, 0, 0, 0]
  Call Extruder 0.02919
  MoveL (T10272) to (120.56, 115.98, 12.3) mm, rotated rx 180 ry 0 rz -180 deg; joints [0, 0, 0, 0, 0, 0]
  Call Extruder 0.02355
  MoveL (T10273) to (119.89, 115.97, 12.3) mm, rotated rx 180 ry 0 rz -180 deg; joints [0, 0, 0, 0, 0, 0]
  Call Extruder 0.02004
  MoveL (T10274) to (120.3, 116.38, 12.3) mm, rotated rx 180 ry 0 rz -180 deg; joints [0, 0, 0, 0, 0, 0]
  Call Extruder 0.02355
  MoveL (T10275) to (119.63, 116.38, 12.3) mm, rotated rx 180 ry 0 rz -180 deg; joints [0, 0, 0, 0, 0, 0]
  Call Extruder 0.01547
  MoveL (T10276) to (119.32, 116.06, 12.3) mm, rotated rx 180 ry 0 rz -180 deg; joints [0, 0, 0, 0, 0, 0]
  Set speed (45.0 mm/s)
  Call Extruder -1.6
  MoveL (T10277) to (119.32, 116.06, 12.3) mm, rotated rx 180 ry 0 rz -180 deg; joints [0, 0, 0, 0, 0, 0]
  Set speed (120.0 mm/s)
  MoveL (T10278) to (119.32, 116.06, 12.3) mm, rotated rx 180 ry 0 rz -180 deg; joints [0, 0, 0, 0, 0, 0]
  Call Extruder -0.15618
  MoveL (T10279) to (119.63, 116.38, 12.3) mm, rotated rx 180 ry 0 rz -180 deg; joints [0, 0, 0, 0, 0, 0]
  Call Extruder -0.22382
  MoveL (T10280) to (120.26, 116.38, 12.3) mm, rotated rx 180 ry 0 rz -180 deg; joints [0, 0, 0, 0, 0, 0]
  Set speed (45.0 mm/s)
  Call Extruder -0.02
  MoveL (T10281) to (120.26, 116.38, 12.3) mm, rotated rx 180 ry 0 rz -180 deg; joints [0, 0, 0, 0, 0, 0]
  Set speed (150.0 mm/s)
  MoveL (T10282) to (120.26, 116.38, 14.3) mm, rotated rx 180 ry 0 rz -180 deg; joints [0, 0, 0, 0, 0, 0]
  MoveL (T10283) to (104.34, 103.54, 14.3) mm, rotated rx 180 ry 0 rz -180 deg; joints [0, 0, 0, 0, 0, 0]
  MoveL (T10284) to (104.34, 103.54, 12.5) mm, rotated rx 180 ry 0 rz -180 deg; joints [0, 0, 0, 0, 0, 0]
  Set speed (40.0 mm/s)
  Call Extruder 2.0
  MoveL (T10285) to (104.34, 103.54, 12.5) mm, rotated rx 180 ry 0 rz -180 deg; joints [0, 0, 0, 0, 0, 0]
  Set speed (25.9 mm/s)
  MoveL (T10286) to (104.34, 103.54, 12.5) mm, rotated rx 180 ry 0 rz -180 deg; joints [0, 0, 0, 0, 0, 0]
  Call Extruder 0.13389
  MoveL (T10287) to (108.73, 103.54, 12.5) mm, rotated rx 180 ry 0 rz -180 deg; joints [0, 0, 0, 0, 0, 0]
  Call Extruder 0.05784
  MoveL (T10288) to (108.73, 105.44, 12.5) mm, rotated rx 180 ry 0 rz -180 deg; joints [0, 0, 0, 0, 0, 0]
  Call Extruder 0.20212
  MoveL (T10289) to (115.37, 105.44, 12.5) mm, rotated rx 180 ry 0 rz -180 deg; joints [0, 0, 0, 0, 0, 0]
  Call Extruder 0.05784
  MoveL (T10290) to (115.37, 103.54, 12.5) mm, rotated rx 180 ry 0 rz -180 deg; joints [0, 0, 0, 0, 0, 0]
  Call Extruder 0.18564
  MoveL (T10291) to (121.46, 103.54, 12.5) mm, rotated rx 180 ry 0 rz -180 deg; joints [0, 0, 0, 0, 0, 0]
  Call Extruder 0.14579
  MoveL (T10292) to (121.46, 108.33, 12.5) mm, rotated rx 180 ry 0 rz -180 deg; joints [0, 0, 0, 0, 0, 0]
  Call Extruder 0.05882
  MoveL (T10293) to (119.53, 108.33, 12.5) mm, rotated rx 180 ry 0 rz -180 deg; joints [0, 0, 0, 0, 0, 0]
  Call Extruder 0.22715
  MoveL (T10294) to (119.53, 115.78, 12.5) mm, rotated rx 180 ry 0 rz -180 deg; joints [0, 0, 0, 0, 0, 0]
  Call Extruder 0.05892
  MoveL (T10295) to (121.46, 115.78, 12.5) mm, rotated rx 180 ry 0 rz -180 deg; joints [0, 0, 0, 0, 0, 0]
  Call Extruder 0.17291
  MoveL (T10296) to (121.46, 121.46, 12.5) mm, rotated rx 180 ry 0 rz -180 deg; joints [0, 0, 0, 0, 0, 0]
  Call Extruder 0.54596
  MoveL (T10297) to (103.54, 121.46, 12.5) mm, rotated rx 180 ry 0 rz -180 deg; joints [0, 0, 0, 0, 0, 0]
  Call Extruder 0.54596
  MoveL (T10298) to (103.54, 103.54, 12.5) mm, rotated rx 180 ry 0 rz -180 deg; joints [0, 0, 0, 0, 0, 0]
  Call Extruder 0.02254
  MoveL (T10299) to (104.28, 103.54, 12.5) mm, rotated rx 180 ry 0 rz -180 deg; joints [0, 0, 0, 0, 0, 0]
  Set speed (150.0 mm/s)
  MoveL (T10300) to (103.53, 103.13, 12.5) mm, rotated rx 180 ry 0 rz -180 deg; joints [0, 0, 0, 0, 0, 0]
  Set speed (25.9 mm/s)
  MoveL (T10301) to (103.53, 103.13, 12.5) mm, rotated rx 180 ry 0 rz -180 deg; joints [0, 0, 0, 0, 0, 0]
  Call Extruder 0.17089
  MoveL (T10302) to (109.14, 103.13, 12.5) mm, rotated rx 180 ry 0 rz -180 deg; joints [0, 0, 0, 0, 0, 0]
  Call Extruder 0.05784
  MoveL (T10303) to (109.14, 105.03, 12.5) mm, rotated rx 180 ry 0 rz -180 deg; joints [0, 0, 0, 0, 0, 0]
  Call Extruder 0.08909
  MoveL (T10304) to (112.06, 105.03, 12.5) mm, rotated rx 180 ry 0 rz -180 deg; joints [0, 0, 0, 0, 0, 0]
  Call Extruder 0.05784
  MoveL (T10305) to (112.07, 103.13, 12.5) mm, rotated rx 180 ry 0 rz -180 deg; joints [0, 0, 0, 0, 0, 0]
  Call Extruder 0.05784
  MoveL (T10306) to (112.08, 105.03, 12.5) mm, rotated rx 180 ry 0 rz -180 deg; joints [0, 0, 0, 0, 0, 0]
  Call Extruder 0.08789
  MoveL (T10307) to (114.96, 105.03, 12.5) mm, rotated rx 180 ry 0 rz -180 deg; joints [0, 0, 0, 0, 0, 0]
  Call Extruder 0.05784
  MoveL (T10308) to (114.96, 103.13, 12.5) mm, rotated rx 180 ry 0 rz -180 deg; joints [0, 0, 0, 0, 0, 0]
  Call Extruder 0.21044
  MoveL (T10309) to (121.87, 103.13, 12.5) mm, rotated rx 180 ry 0 rz -180 deg; joints [0, 0, 0, 0, 0, 0]
  Call Extruder 0.17059
  MoveL (T10310) to (121.87, 108.73, 12.5) mm, rotated rx 180 ry 0 rz -180 deg; joints [0, 0, 0, 0, 0, 0]
  Call Extruder 0.05882
  MoveL (T10311) to (119.94, 108.73, 12.5) mm, rotated rx 180 ry 0 rz -180 deg; joints [0, 0, 0, 0, 0, 0]
  Call Extruder 0.09013
  MoveL (T10312) to (119.94, 111.69, 12.5) mm, rotated rx 180 ry 0 rz -180 deg; joints [0, 0, 0, 0, 0, 0]
  Call Extruder 0.05886
  MoveL (T10313) to (121.87, 111.69, 12.5) mm, rotated rx 180 ry 0 rz -180 deg; joints [0, 0, 0, 0, 0, 0]
  Call Extruder 0.0226
  MoveL (T10314) to (121.87, 112.43, 12.5) mm, rotated rx 180 ry 0 rz -180 deg; joints [0, 0, 0, 0, 0, 0]
  Call Extruder 0.05887
  MoveL (T10315) to (119.94, 112.43, 12.5) mm, rotated rx 180 ry 0 rz -180 deg; joints [0, 0, 0, 0, 0, 0]
  Call Extruder 0.08975
  MoveL (T10316) to (119.93, 115.38, 12.5) mm, rotated rx 180 ry 0 rz -180 deg; joints [0, 0, 0, 0, 0, 0]
  Call Extruder 0.05891
  MoveL (T10317) to (121.87, 115.38, 12.5) mm, rotated rx 180 ry 0 rz -180 deg; joints [0, 0, 0, 0, 0, 0]
  Call Extruder 0.1977
  MoveL (T10318) to (121.87, 121.87, 12.5) mm, rotated rx 180 ry 0 rz -180 deg; joints [0, 0, 0, 0, 0, 0]
  Call Extruder 0.57077
  MoveL (T10319) to (103.13, 121.87, 12.5) mm, rotated rx 180 ry 0 rz -180 deg; joints [0, 0, 0, 0, 0, 0]
  Call Extruder 0.57077
  MoveL (T10320) to (103.13, 103.13, 12.5) mm, rotated rx 180 ry 0 rz -180 deg; joints [0, 0, 0, 0, 0, 0]
  Call Extruder 0.01036
  MoveL (T10321) to (103.47, 103.13, 12.5) mm, rotated rx 180 ry 0 rz -180 deg; joints [0, 0, 0, 0, 0, 0]
  Set speed (150.0 mm/s)
  MoveL (T10322) to (102.72, 102.81, 12.5) mm, rotated rx 180 ry 0 rz -180 deg; joints [0, 0, 0, 0, 0, 0]
  Set speed (25.0 mm/s)
  MoveL (T10323) to (102.72, 102.81, 12.5) mm, rotated rx 180 ry 0 rz -180 deg; joints [0, 0, 0, 0, 0, 0]
  Call Extruder 0.00259
  MoveL (T10324) to (102.72, 102.72, 12.5) mm, rotated rx 180 ry 0 rz -180 deg; joints [0, 0, 0, 0, 0, 0]
  Call Extruder 0.20788
  MoveL (T10325) to (109.55, 102.72, 12.5) mm, rotated rx 180 ry 0 rz -180 deg; joints [0, 0, 0, 0, 0, 0]
  Call Extruder 0.05784
  MoveL (T10326) to (109.55, 104.62, 12.5) mm, rotated rx 180 ry 0 rz -180 deg; joints [0, 0, 0, 0, 0, 0]
  Call Extruder 0.06429
  MoveL (T10327) to (111.66, 104.62, 12.5) mm, rotated rx 180 ry 0 rz -180 deg; joints [0, 0, 0, 0, 0, 0]
  Call Extruder 0.05784
  MoveL (T10328) to (111.66, 102.72, 12.5) mm, rotated rx 180 ry 0 rz -180 deg; joints [0, 0, 0, 0, 0, 0]
  Call Extruder 0.02506
  MoveL (T10329) to (112.48, 102.72, 12.5) mm, rotated rx 180 ry 0 rz -180 deg; joints [0, 0, 0, 0, 0, 0]
  Call Extruder 0.05784
  MoveL (T10330) to (112.48, 104.62, 12.5) mm, rotated rx 180 ry 0 rz -180 deg; joints [0, 0, 0, 0, 0, 0]
  Call Extruder 0.06309
  MoveL (T10331) to (114.55, 104.62, 12.5) mm, rotated rx 180 ry 0 rz -180 deg; joints [0, 0, 0, 0, 0, 0]
  Call Extruder 0.05784
  MoveL (T10332) to (114.55, 102.72, 12.5) mm, rotated rx 180 ry 0 rz -180 deg; joints [0, 0, 0, 0, 0, 0]
  Call Extruder 0.23525
  MoveL (T10333) to (122.28, 102.72, 12.5) mm, rotated rx 180 ry 0 rz -180 deg; joints [0, 0, 0, 0, 0, 0]
  Call Extruder 0.19539
  MoveL (T10334) to (122.28, 109.14, 12.5) mm, rotated rx 180 ry 0 rz -180 deg; joints [0, 0, 0, 0, 0, 0]
  Call Extruder 0.05883
  MoveL (T10335) to (120.34, 109.14, 12.5) mm, rotated rx 180 ry 0 rz -180 deg; joints [0, 0, 0, 0, 0, 0]
  Call Extruder 0.06533
  MoveL (T10336) to (120.34, 111.28, 12.5) mm, rotated rx 180 ry 0 rz -180 deg; joints [0, 0, 0, 0, 0, 0]
  Call Extruder 0.05886
  MoveL (T10337) to (122.28, 111.28, 12.5) mm, rotated rx 180 ry 0 rz -180 deg; joints [0, 0, 0, 0, 0, 0]
  Call Extruder 0.04742
  MoveL (T10338) to (122.28, 112.84, 12.5) mm, rotated rx 180 ry 0 rz -180 deg; joints [0, 0, 0, 0, 0, 0]
  Call Extruder 0.05888
  MoveL (T10339) to (120.34, 112.84, 12.5) mm, rotated rx 180 ry 0 rz -180 deg; joints [0, 0, 0, 0, 0, 0]
  Call Extruder 0.06495
  MoveL (T10340) to (120.34, 114.97, 12.5) mm, rotated rx 180 ry 0 rz -180 deg; joints [0, 0, 0, 0, 0, 0]
  Call Extruder 0.05891
  MoveL (T10341) to (122.28, 114.97, 12.5) mm, rotated rx 180 ry 0 rz -180 deg; joints [0, 0, 0, 0, 0, 0]
  Call Extruder 0.22249
  MoveL (T10342) to (122.28, 122.28, 12.5) mm, rotated rx 180 ry 0 rz -180 deg; joints [0, 0, 0, 0, 0, 0]
  Call Extruder 0.59557
  MoveL (T10343) to (102.72, 122.28, 12.5) mm, rotated rx 180 ry 0 rz -180 deg; joints [0, 0, 0, 0, 0, 0]
  Call Extruder 0.59115
  MoveL (T10344) to (102.72, 102.87, 12.5) mm, rotated rx 180 ry 0 rz -180 deg; joints [0, 0, 0, 0, 0, 0]
  Set speed (150.0 mm/s)
  MoveL (T10345) to (102.78, 102.75, 12.5) mm, rotated rx 180 ry 0 rz -180 deg; joints [0, 0, 0, 0, 0, 0]
  Set speed (45.0 mm/s)
  Call Extruder -1.6
  MoveL (T10346) to (102.78, 102.75, 12.5) mm, rotated rx 180 ry 0 rz -180 deg; joints [0, 0, 0, 0, 0, 0]
  Set speed (120.0 mm/s)
  MoveL (T10347) to (102.78, 102.75, 12.5) mm, rotated rx 180 ry 0 rz -180 deg; joints [0, 0, 0, 0, 0, 0]
  Call Extruder -0.05166
  MoveL (T10348) to (102.72, 102.72, 12.5) mm, rotated rx 180 ry 0 rz -180 deg; joints [0, 0, 0, 0, 0, 0]
  Call Extruder -0.32834
  MoveL (T10349) to (103.65, 102.72, 12.5) mm, rotated rx 180 ry 0 rz -180 deg; joints [0, 0, 0, 0, 0, 0]
  Set speed (45.0 mm/s)
  Call Extruder -0.02
  MoveL (T10350) to (103.65, 102.72, 12.5) mm, rotated rx 180 ry 0 rz -180 deg; joints [0, 0, 0, 0, 0, 0]
  Set speed (150.0 mm/s)
  MoveL (T10351) to (103.65, 102.72, 14.5) mm, rotated rx 180 ry 0 rz -180 deg; joints [0, 0, 0, 0, 0, 0]
  MoveL (T10352) to (106.29, 103.84, 14.5) mm, rotated rx 180 ry 0 rz -180 deg; joints [0, 0, 0, 0, 0, 0]
  MoveL (T10353) to (106.29, 103.84, 12.5) mm, rotated rx 180 ry 0 rz -180 deg; joints [0, 0, 0, 0, 0, 0]
  Set speed (40.0 mm/s)
  Call Extruder 2.0
  MoveL (T10354) to (106.29, 103.84, 12.5) mm, rotated rx 180 ry 0 rz -180 deg; joints [0, 0, 0, 0, 0, 0]
  Set speed (25.9 mm/s)
  MoveL (T10355) to (106.29, 103.84, 12.5) mm, rotated rx 180 ry 0 rz -180 deg; joints [0, 0, 0, 0, 0, 0]
  Call Extruder 0.07441
  MoveL (T10356) to (103.84, 103.84, 12.5) mm, rotated rx 180 ry 0 rz -180 deg; joints [0, 0, 0, 0, 0, 0]
  Call Extruder 0.7458
  MoveL (T10357) to (121.16, 121.16, 12.5) mm, rotated rx 180 ry 0 rz -180 deg; joints [0, 0, 0, 0, 0, 0]
  Call Extruder 0.10645
  MoveL (T10358) to (121.16, 117.66, 12.5) mm, rotated rx 180 ry 0 rz -180 deg; joints [0, 0, 0, 0, 0, 0]
  Call Extruder 0.15054
  MoveL (T10359) to (117.66, 121.16, 12.5) mm, rotated rx 180 ry 0 rz -180 deg; joints [0, 0, 0, 0, 0, 0]
  Call Extruder 0.03385
  MoveL (T10360) to (116.55, 121.16, 12.5) mm, rotated rx 180 ry 0 rz -180 deg; joints [0, 0, 0, 0, 0, 0]
  Call Extruder 0.54738
  MoveL (T10361) to (103.84, 108.45, 12.5) mm, rotated rx 180 ry 0 rz -180 deg; joints [0, 0, 0, 0, 0, 0]
  Call Extruder 0.03385
  MoveL (T10362) to (103.84, 107.34, 12.5) mm, rotated rx 180 ry 0 rz -180 deg; joints [0, 0, 0, 0, 0, 0]
  Call Extruder 0.15054
  MoveL (T10363) to (107.34, 103.84, 12.5) mm, rotated rx 180 ry 0 rz -180 deg; joints [0, 0, 0, 0, 0, 0]
  Call Extruder 0.00874
  MoveL (T10364) to (107.63, 103.84, 12.5) mm, rotated rx 180 ry 0 rz -180 deg; joints [0, 0, 0, 0, 0, 0]
  Call Extruder 0.05204
  MoveL (T10365) to (107.62, 105.55, 12.5) mm, rotated rx 180 ry 0 rz -180 deg; joints [0, 0, 0, 0, 0, 0]
  Call Extruder 0.01363
  MoveL (T10366) to (107.94, 105.87, 12.5) mm, rotated rx 180 ry 0 rz -180 deg; joints [0, 0, 0, 0, 0, 0]
  Set speed (150.0 mm/s)
  MoveL (T10367) to (108.61, 105.28, 12.5) mm, rotated rx 180 ry 0 rz -180 deg; joints [0, 0, 0, 0, 0, 0]
  Set speed (25.9 mm/s)
  MoveL (T10368) to (108.61, 105.28, 12.5) mm, rotated rx 180 ry 0 rz -180 deg; joints [0, 0, 0, 0, 0, 0]
  Call Extruder 0.00925
  MoveL (T10369) to (108.43, 105.47, 12.5) mm, rotated rx 180 ry 0 rz -180 deg; joints [0, 0, 0, 0, 0, 0]
  Call Extruder 0.01116
  MoveL (T10370) to (108.11, 105.47, 12.5) mm, rotated rx 180 ry 0 rz -180 deg; joints [0, 0, 0, 0, 0, 0]
  Call Extruder 0.00408
  MoveL (T10371) to (108.03, 105.38, 12.5) mm, rotated rx 180 ry 0 rz -180 deg; joints [0, 0, 0, 0, 0, 0]
  Call Extruder 0.00694
  MoveL (T10372) to (108.03, 105.19, 12.5) mm, rotated rx 180 ry 0 rz -180 deg; joints [0, 0, 0, 0, 0, 0]
  Call Extruder 0.01991
  MoveL (T10373) to (108.43, 104.79, 12.5) mm, rotated rx 180 ry 0 rz -180 deg; joints [0, 0, 0, 0, 0, 0]
  Call Extruder 0.02387
  MoveL (T10374) to (108.43, 104.12, 12.5) mm, rotated rx 180 ry 0 rz -180 deg; joints [0, 0, 0, 0, 0, 0]
  Call Extruder 0.01991
  MoveL (T10375) to (108.03, 104.52, 12.5) mm, rotated rx 180 ry 0 rz -180 deg; joints [0, 0, 0, 0, 0, 0]
  Call Extruder 0.02387
  MoveL (T10376) to (108.03, 103.84, 12.5) mm, rotated rx 180 ry 0 rz -180 deg; joints [0, 0, 0, 0, 0, 0]
  Call Extruder 0.00924
  MoveL (T10377) to (108.22, 103.66, 12.5) mm, rotated rx 180 ry 0 rz -180 deg; joints [0, 0, 0, 0, 0, 0]
  Set speed (45.0 mm/s)
  Call Extruder -1.6
  MoveL (T10378) to (108.22, 103.66, 12.5) mm, rotated rx 180 ry 0 rz -180 deg; joints [0, 0, 0, 0, 0, 0]
  Set speed (120.0 mm/s)
  MoveL (T10379) to (108.22, 103.66, 12.5) mm, rotated rx 180 ry 0 rz -180 deg; joints [0, 0, 0, 0, 0, 0]
  Call Extruder -0.09262
  MoveL (T10380) to (108.03, 103.84, 12.5) mm, rotated rx 180 ry 0 rz -180 deg; joints [0, 0, 0, 0, 0, 0]
  Call Extruder -0.23934
  MoveL (T10381) to (108.03, 104.52, 12.5) mm, rotated rx 180 ry 0 rz -180 deg; joints [0, 0, 0, 0, 0, 0]
  Call Extruder -0.04804
  MoveL (T10382) to (108.13, 104.42, 12.5) mm, rotated rx 180 ry 0 rz -180 deg; joints [0, 0, 0, 0, 0, 0]
  Set speed (45.0 mm/s)
  Call Extruder -0.02
  MoveL (T10383) to (108.13, 104.42, 12.5) mm, rotated rx 180 ry 0 rz -180 deg; joints [0, 0, 0, 0, 0, 0]
  Set speed (150.0 mm/s)
  MoveL (T10384) to (108.13, 104.42, 14.5) mm, rotated rx 180 ry 0 rz -180 deg; joints [0, 0, 0, 0, 0, 0]
  MoveL (T10385) to (103.84, 109.5, 14.5) mm, rotated rx 180 ry 0 rz -180 deg; joints [0, 0, 0, 0, 0, 0]
  MoveL (T10386) to (103.84, 109.5, 12.5) mm, rotated rx 180 ry 0 rz -180 deg; joints [0, 0, 0, 0, 0, 0]
  Set speed (40.0 mm/s)
  Call Extruder 2.0
  MoveL (T10387) to (103.84, 109.5, 12.5) mm, rotated rx 180 ry 0 rz -180 deg; joints [0, 0, 0, 0, 0, 0]
  Set speed (25.9 mm/s)
  MoveL (T10388) to (103.84, 109.5, 12.5) mm, rotated rx 180 ry 0 rz -180 deg; joints [0, 0, 0, 0, 0, 0]
  Call Extruder 0.07441
  MoveL (T10389) to (103.84, 111.94, 12.5) mm, rotated rx 180 ry 0 rz -180 deg; joints [0, 0, 0, 0, 0, 0]
  Call Extruder 0.26717
  MoveL (T10390) to (110.05, 105.74, 12.5) mm, rotated rx 180 ry 0 rz -180 deg; joints [0, 0, 0, 0, 0, 0]
  Call Extruder 0.00923
  MoveL (T10391) to (110.35, 105.74, 12.5) mm, rotated rx 180 ry 0 rz -180 deg; joints [0, 0, 0, 0, 0, 0]
  Call Extruder 0.38229
  MoveL (T10392) to (119.22, 114.62, 12.5) mm, rotated rx 180 ry 0 rz -180 deg; joints [0, 0, 0, 0, 0, 0]
  Call Extruder 0.01136
  MoveL (T10393) to (119.22, 114.99, 12.5) mm, rotated rx 180 ry 0 rz -180 deg; joints [0, 0, 0, 0, 0, 0]
  Call Extruder 0.26565
  MoveL (T10394) to (113.06, 121.16, 12.5) mm, rotated rx 180 ry 0 rz -180 deg; joints [0, 0, 0, 0, 0, 0]
  Call Extruder 0.03385
  MoveL (T10395) to (111.94, 121.16, 12.5) mm, rotated rx 180 ry 0 rz -180 deg; joints [0, 0, 0, 0, 0, 0]
  Call Extruder 0.34896
  MoveL (T10396) to (103.84, 113.06, 12.5) mm, rotated rx 180 ry 0 rz -180 deg; joints [0, 0, 0, 0, 0, 0]
  Call Extruder 0.10645
  MoveL (T10397) to (103.84, 116.55, 12.5) mm, rotated rx 180 ry 0 rz -180 deg; joints [0, 0, 0, 0, 0, 0]
  Call Extruder 0.46559
  MoveL (T10398) to (114.65, 105.74, 12.5) mm, rotated rx 180 ry 0 rz -180 deg; joints [0, 0, 0, 0, 0, 0]
  Call Extruder 0.00923
  MoveL (T10399) to (114.95, 105.74, 12.5) mm, rotated rx 180 ry 0 rz -180 deg; joints [0, 0, 0, 0, 0, 0]
  Call Extruder 0.18395
  MoveL (T10400) to (119.22, 110.01, 12.5) mm, rotated rx 180 ry 0 rz -180 deg; joints [0, 0, 0, 0, 0, 0]
  Call Extruder 0.01124
  MoveL (T10401) to (119.22, 110.38, 12.5) mm, rotated rx 180 ry 0 rz -180 deg; joints [0, 0, 0, 0, 0, 0]
  Call Extruder 0.46416
  MoveL (T10402) to (108.45, 121.16, 12.5) mm, rotated rx 180 ry 0 rz -180 deg; joints [0, 0, 0, 0, 0, 0]
  Call Extruder 0.03385
  MoveL (T10403) to (107.34, 121.16, 12.5) mm, rotated rx 180 ry 0 rz -180 deg; joints [0, 0, 0, 0, 0, 0]
  Call Extruder 0.15054
  MoveL (T10404) to (103.84, 117.66, 12.5) mm, rotated rx 180 ry 0 rz -180 deg; joints [0, 0, 0, 0, 0, 0]
  Call Extruder 0.10645
  MoveL (T10405) to (103.84, 121.16, 12.5) mm, rotated rx 180 ry 0 rz -180 deg; joints [0, 0, 0, 0, 0, 0]
  Call Extruder 0.7458
  MoveL (T10406) to (121.16, 103.84, 12.5) mm, rotated rx 180 ry 0 rz -180 deg; joints [0, 0, 0, 0, 0, 0]
  Call Extruder 0.10143
  MoveL (T10407) to (121.16, 107.17, 12.5) mm, rotated rx 180 ry 0 rz -180 deg; joints [0, 0, 0, 0, 0, 0]
  Call Extruder 0.00502
  MoveL (T10408) to (120.99, 107.17, 12.5) mm, rotated rx 180 ry 0 rz -180 deg; joints [0, 0, 0, 0, 0, 0]
  Call Extruder 0.14344
  MoveL (T10409) to (117.66, 103.84, 12.5) mm, rotated rx 180 ry 0 rz -180 deg; joints [0, 0, 0, 0, 0, 0]
  Call Extruder 0.0333
  MoveL (T10410) to (116.57, 103.84, 12.5) mm, rotated rx 180 ry 0 rz -180 deg; joints [0, 0, 0, 0, 0, 0]
  Call Extruder 0.0411
  MoveL (T10411) to (116.57, 105.19, 12.5) mm, rotated rx 180 ry 0 rz -180 deg; joints [0, 0, 0, 0, 0, 0]
  Set speed (150.0 mm/s)
  MoveL (T10412) to (115.84, 105.65, 12.5) mm, rotated rx 180 ry 0 rz -180 deg; joints [0, 0, 0, 0, 0, 0]
  Set speed (25.9 mm/s)
  MoveL (T10413) to (115.84, 105.65, 12.5) mm, rotated rx 180 ry 0 rz -180 deg; joints [0, 0, 0, 0, 0, 0]
  Call Extruder 0.01615
  MoveL (T10414) to (116.16, 105.33, 12.5) mm, rotated rx 180 ry 0 rz -180 deg; joints [0, 0, 0, 0, 0, 0]
  Call Extruder 0.02452
  MoveL (T10415) to (116.16, 104.65, 12.5) mm, rotated rx 180 ry 0 rz -180 deg; joints [0, 0, 0, 0, 0, 0]
  Call Extruder 0.02486
  MoveL (T10416) to (115.67, 105.14, 12.5) mm, rotated rx 180 ry 0 rz -180 deg; joints [0, 0, 0, 0, 0, 0]
  Call Extruder 0.02452
  MoveL (T10417) to (115.67, 104.46, 12.5) mm, rotated rx 180 ry 0 rz -180 deg; joints [0, 0, 0, 0, 0, 0]
  Call Extruder 0.03419
  MoveL (T10418) to (116.34, 103.79, 12.5) mm, rotated rx 180 ry 0 rz -180 deg; joints [0, 0, 0, 0, 0, 0]
  Set speed (45.0 mm/s)
  Call Extruder -1.6
  MoveL (T10419) to (116.34, 103.79, 12.5) mm, rotated rx 180 ry 0 rz -180 deg; joints [0, 0, 0, 0, 0, 0]
  Set speed (120.0 mm/s)
  MoveL (T10420) to (116.34, 103.79, 12.5) mm, rotated rx 180 ry 0 rz -180 deg; joints [0, 0, 0, 0, 0, 0]
  Call Extruder -0.33806
  MoveL (T10421) to (115.67, 104.46, 12.5) mm, rotated rx 180 ry 0 rz -180 deg; joints [0, 0, 0, 0, 0, 0]
  Call Extruder -0.04194
  MoveL (T10422) to (115.67, 104.58, 12.5) mm, rotated rx 180 ry 0 rz -180 deg; joints [0, 0, 0, 0, 0, 0]
  Set speed (45.0 mm/s)
  Call Extruder -0.02
  MoveL (T10423) to (115.67, 104.58, 12.5) mm, rotated rx 180 ry 0 rz -180 deg; joints [0, 0, 0, 0, 0, 0]
  Set speed (150.0 mm/s)
  MoveL (T10424) to (115.67, 104.58, 14.5) mm, rotated rx 180 ry 0 rz -180 deg; joints [0, 0, 0, 0, 0, 0]
  MoveL (T10425) to (121.17, 107.4, 14.5) mm, rotated rx 180 ry 0 rz -180 deg; joints [0, 0, 0, 0, 0, 0]
  MoveL (T10426) to (121.17, 107.4, 12.5) mm, rotated rx 180 ry 0 rz -180 deg; joints [0, 0, 0, 0, 0, 0]
  Set speed (40.0 mm/s)
  Call Extruder 2.0
  MoveL (T10427) to (121.17, 107.4, 12.5) mm, rotated rx 180 ry 0 rz -180 deg; joints [0, 0, 0, 0, 0, 0]
  Set speed (25.9 mm/s)
  MoveL (T10428) to (121.17, 107.4, 12.5) mm, rotated rx 180 ry 0 rz -180 deg; joints [0, 0, 0, 0, 0, 0]
  Call Extruder 0.03146
  MoveL (T10429) to (120.55, 108.02, 12.5) mm, rotated rx 180 ry 0 rz -180 deg; joints [0, 0, 0, 0, 0, 0]
  Call Extruder 0.02417
  MoveL (T10430) to (119.87, 108.02, 12.5) mm, rotated rx 180 ry 0 rz -180 deg; joints [0, 0, 0, 0, 0, 0]
  Call Extruder 0.0222
  MoveL (T10431) to (120.31, 107.58, 12.5) mm, rotated rx 180 ry 0 rz -180 deg; joints [0, 0, 0, 0, 0, 0]
  Call Extruder 0.02417
  MoveL (T10432) to (119.64, 107.58, 12.5) mm, rotated rx 180 ry 0 rz -180 deg; joints [0, 0, 0, 0, 0, 0]
  Call Extruder 0.0159
  MoveL (T10433) to (119.32, 107.9, 12.5) mm, rotated rx 180 ry 0 rz -180 deg; joints [0, 0, 0, 0, 0, 0]
  Set speed (45.0 mm/s)
  Call Extruder -1.6
  MoveL (T10434) to (119.32, 107.9, 12.5) mm, rotated rx 180 ry 0 rz -180 deg; joints [0, 0, 0, 0, 0, 0]
  Set speed (120.0 mm/s)
  MoveL (T10435) to (119.32, 107.9, 12.5) mm, rotated rx 180 ry 0 rz -180 deg; joints [0, 0, 0, 0, 0, 0]
  Call Extruder -0.15842
  MoveL (T10436) to (119.64, 107.58, 12.5) mm, rotated rx 180 ry 0 rz -180 deg; joints [0, 0, 0, 0, 0, 0]
  Call Extruder -0.22158
  MoveL (T10437) to (120.26, 107.58, 12.5) mm, rotated rx 180 ry 0 rz -180 deg; joints [0, 0, 0, 0, 0, 0]
  Set speed (45.0 mm/s)
  Call Extruder -0.02
  MoveL (T10438) to (120.26, 107.58, 12.5) mm, rotated rx 180 ry 0 rz -180 deg; joints [0, 0, 0, 0, 0, 0]
  Set speed (150.0 mm/s)
  MoveL (T10439) to (120.26, 107.58, 14.5) mm, rotated rx 180 ry 0 rz -180 deg; joints [0, 0, 0, 0, 0, 0]
  MoveL (T10440) to (119.73, 112.06, 14.5) mm, rotated rx 180 ry 0 rz -180 deg; joints [0, 0, 0, 0, 0, 0]
  MoveL (T10441) to (119.73, 112.06, 12.5) mm, rotated rx 180 ry 0 rz -180 deg; joints [0, 0, 0, 0, 0, 0]
  Set speed (40.0 mm/s)
  Call Extruder 2.0
  MoveL (T10442) to (119.73, 112.06, 12.5) mm, rotated rx 180 ry 0 rz -180 deg; joints [0, 0, 0, 0, 0, 0]
  Set speed (25.9 mm/s)
  MoveL (T10443) to (119.73, 112.06, 12.5) mm, rotated rx 180 ry 0 rz -180 deg; joints [0, 0, 0, 0, 0, 0]
  Call Extruder 0.0483
  MoveL (T10444) to (121.66, 112.06, 12.5) mm, rotated rx 180 ry 0 rz -180 deg; joints [0, 0, 0, 0, 0, 0]
  Set speed (45.0 mm/s)
  Call Extruder -1.6
  MoveL (T10445) to (121.66, 112.06, 12.5) mm, rotated rx 180 ry 0 rz -180 deg; joints [0, 0, 0, 0, 0, 0]
  Set speed (120.0 mm/s)
  MoveL (T10446) to (121.66, 112.06, 12.5) mm, rotated rx 180 ry 0 rz -180 deg; joints [0, 0, 0, 0, 0, 0]
  Call Extruder -0.38
  MoveL (T10447) to (120.6, 112.06, 12.5) mm, rotated rx 180 ry 0 rz -180 deg; joints [0, 0, 0, 0, 0, 0]
  Set speed (45.0 mm/s)
  Call Extruder -0.02
  MoveL (T10448) to (120.6, 112.06, 12.5) mm, rotated rx 180 ry 0 rz -180 deg; joints [0, 0, 0, 0, 0, 0]
  Set speed (150.0 mm/s)
  MoveL (T10449) to (120.6, 112.06, 14.5) mm, rotated rx 180 ry 0 rz -180 deg; joints [0, 0, 0, 0, 0, 0]
  MoveL (T10450) to (121.34, 116.3, 14.5) mm, rotated rx 180 ry 0 rz -180 deg; joints [0, 0, 0, 0, 0, 0]
  MoveL (T10451) to (121.34, 116.3, 12.5) mm, rotated rx 180 ry 0 rz -180 deg; joints [0, 0, 0, 0, 0, 0]
  Set speed (40.0 mm/s)
  Call Extruder 2.0
  MoveL (T10452) to (121.34, 116.3, 12.5) mm, rotated rx 180 ry 0 rz -180 deg; joints [0, 0, 0, 0, 0, 0]
  Set speed (25.9 mm/s)
  MoveL (T10453) to (121.34, 116.3, 12.5) mm, rotated rx 180 ry 0 rz -180 deg; joints [0, 0, 0, 0, 0, 0]
  Call Extruder 0.00966
  MoveL (T10454) to (121.15, 116.49, 12.5) mm, rotated rx 180 ry 0 rz -180 deg; joints [0, 0, 0, 0, 0, 0]
  Call Extruder 0.02457
  MoveL (T10455) to (120.47, 116.49, 12.5) mm, rotated rx 180 ry 0 rz -180 deg; joints [0, 0, 0, 0, 0, 0]
  Call Extruder 0.02044
  MoveL (T10456) to (120.87, 116.09, 12.5) mm, rotated rx 180 ry 0 rz -180 deg; joints [0, 0, 0, 0, 0, 0]
  Call Extruder 0.02457
  MoveL (T10457) to (120.19, 116.09, 12.5) mm, rotated rx 180 ry 0 rz -180 deg; joints [0, 0, 0, 0, 0, 0]
  Call Extruder 0.02044
  MoveL (T10458) to (119.79, 116.49, 12.5) mm, rotated rx 180 ry 0 rz -180 deg; joints [0, 0, 0, 0, 0, 0]
  Call Extruder 0.00739
  MoveL (T10459) to (119.58, 116.49, 12.5) mm, rotated rx 180 ry 0 rz -180 deg; joints [0, 0, 0, 0, 0, 0]
  Call Extruder 0.00413
  MoveL (T10460) to (119.5, 116.41, 12.5) mm, rotated rx 180 ry 0 rz -180 deg; joints [0, 0, 0, 0, 0, 0]
  Call Extruder 0.01134
  MoveL (T10461) to (119.5, 116.09, 12.5) mm, rotated rx 180 ry 0 rz -180 deg; joints [0, 0, 0, 0, 0, 0]
  Call Extruder 0.00964
  MoveL (T10462) to (119.69, 115.91, 12.5) mm, rotated rx 180 ry 0 rz -180 deg; joints [0, 0, 0, 0, 0, 0]
  Set speed (45.0 mm/s)
  Call Extruder -1.6
  MoveL (T10463) to (119.69, 115.91, 12.5) mm, rotated rx 180 ry 0 rz -180 deg; joints [0, 0, 0, 0, 0, 0]
  Set speed (120.0 mm/s)
  MoveL (T10464) to (119.69, 115.91, 12.5) mm, rotated rx 180 ry 0 rz -180 deg; joints [0, 0, 0, 0, 0, 0]
  Call Extruder -0.09521
  MoveL (T10465) to (119.5, 116.09, 12.5) mm, rotated rx 180 ry 0 rz -180 deg; joints [0, 0, 0, 0, 0, 0]
  Call Extruder -0.11197
  MoveL (T10466) to (119.5, 116.41, 12.5) mm, rotated rx 180 ry 0 rz -180 deg; joints [0, 0, 0, 0, 0, 0]
  Call Extruder -0.04075
  MoveL (T10467) to (119.58, 116.49, 12.5) mm, rotated rx 180 ry 0 rz -180 deg; joints [0, 0, 0, 0, 0, 0]
  Call Extruder -0.07298
  MoveL (T10468) to (119.79, 116.49, 12.5) mm, rotated rx 180 ry 0 rz -180 deg; joints [0, 0, 0, 0, 0, 0]
  Call Extruder -0.0591
  MoveL (T10469) to (119.91, 116.37, 12.5) mm, rotated rx 180 ry 0 rz -180 deg; joints [0, 0, 0, 0, 0, 0]
  Set speed (45.0 mm/s)
  Call Extruder -0.02
  MoveL (T10470) to (119.91, 116.37, 12.5) mm, rotated rx 180 ry 0 rz -180 deg; joints [0, 0, 0, 0, 0, 0]
  Set speed (150.0 mm/s)
  MoveL (T10471) to (119.91, 116.37, 14.5) mm, rotated rx 180 ry 0 rz -180 deg; joints [0, 0, 0, 0, 0, 0]
  MoveL (T10472) to (104.34, 103.54, 14.5) mm, rotated rx 180 ry 0 rz -180 deg; joints [0, 0, 0, 0, 0, 0]
  MoveL (T10473) to (104.34, 103.54, 12.7) mm, rotated rx 180 ry 0 rz -180 deg; joints [0, 0, 0, 0, 0, 0]
  Set speed (40.0 mm/s)
  Call Extruder 2.0
  MoveL (T10474) to (104.34, 103.54, 12.7) mm, rotated rx 180 ry 0 rz -180 deg; joints [0, 0, 0, 0, 0, 0]
  Set speed (26.0 mm/s)
  MoveL (T10475) to (104.34, 103.54, 12.7) mm, rotated rx 180 ry 0 rz -180 deg; joints [0, 0, 0, 0, 0, 0]
  Call Extruder 0.13047
  MoveL (T10476) to (108.62, 103.54, 12.7) mm, rotated rx 180 ry 0 rz -180 deg; joints [0, 0, 0, 0, 0, 0]
  Call Extruder 0.05784
  MoveL (T10477) to (108.62, 105.44, 12.7) mm, rotated rx 180 ry 0 rz -180 deg; joints [0, 0, 0, 0, 0, 0]
  Call Extruder 0.0967
  MoveL (T10478) to (111.8, 105.44, 12.7) mm, rotated rx 180 ry 0 rz -180 deg; joints [0, 0, 0, 0, 0, 0]
  Call Extruder 0.11274
  MoveL (T10479) to (115.5, 105.44, 12.7) mm, rotated rx 180 ry 0 rz -180 deg; joints [0, 0, 0, 0, 0, 0]
  Call Extruder 0.05784
  MoveL (T10480) to (115.5, 103.54, 12.7) mm, rotated rx 180 ry 0 rz -180 deg; joints [0, 0, 0, 0, 0, 0]
  Call Extruder 0.18174
  MoveL (T10481) to (121.46, 103.54, 12.7) mm, rotated rx 180 ry 0 rz -180 deg; joints [0, 0, 0, 0, 0, 0]
  Call Extruder 0.14215
  MoveL (T10482) to (121.46, 108.2, 12.7) mm, rotated rx 180 ry 0 rz -180 deg; joints [0, 0, 0, 0, 0, 0]
  Call Extruder 0.05881
  MoveL (T10483) to (119.53, 108.21, 12.7) mm, rotated rx 180 ry 0 rz -180 deg; joints [0, 0, 0, 0, 0, 0]
  Call Extruder 0.11502
  MoveL (T10484) to (119.53, 111.98, 12.7) mm, rotated rx 180 ry 0 rz -180 deg; joints [0, 0, 0, 0, 0, 0]
  Call Extruder 0.05886
  MoveL (T10485) to (121.46, 111.98, 12.7) mm, rotated rx 180 ry 0 rz -180 deg; joints [0, 0, 0, 0, 0, 0]
  Call Extruder 0.00472
  MoveL (T10486) to (121.46, 112.14, 12.7) mm, rotated rx 180 ry 0 rz -180 deg; joints [0, 0, 0, 0, 0, 0]
  Call Extruder 0.05886
  MoveL (T10487) to (119.53, 112.13, 12.7) mm, rotated rx 180 ry 0 rz -180 deg; joints [0, 0, 0, 0, 0, 0]
  Call Extruder 0.11462
  MoveL (T10488) to (119.53, 115.9, 12.7) mm, rotated rx 180 ry 0 rz -180 deg; joints [0, 0, 0, 0, 0, 0]
  Call Extruder 0.05891
  MoveL (T10489) to (121.46, 115.9, 12.7) mm, rotated rx 180 ry 0 rz -180 deg; joints [0, 0, 0, 0, 0, 0]
  Call Extruder 0.16946
  MoveL (T10490) to (121.46, 121.46, 12.7) mm, rotated rx 180 ry 0 rz -180 deg; joints [0, 0, 0, 0, 0, 0]
  Call Extruder 0.54596
  MoveL (T10491) to (103.54, 121.46, 12.7) mm, rotated rx 180 ry 0 rz -180 deg; joints [0, 0, 0, 0, 0, 0]
  Call Extruder 0.54596
  MoveL (T10492) to (103.54, 103.54, 12.7) mm, rotated rx 180 ry 0 rz -180 deg; joints [0, 0, 0, 0, 0, 0]
  Call Extruder 0.02254
  MoveL (T10493) to (104.28, 103.54, 12.7) mm, rotated rx 180 ry 0 rz -180 deg; joints [0, 0, 0, 0, 0, 0]
  Set speed (150.0 mm/s)
  MoveL (T10494) to (103.53, 103.13, 12.7) mm, rotated rx 180 ry 0 rz -180 deg; joints [0, 0, 0, 0, 0, 0]
  Set speed (26.0 mm/s)
  MoveL (T10495) to (103.53, 103.13, 12.7) mm, rotated rx 180 ry 0 rz -180 deg; joints [0, 0, 0, 0, 0, 0]
  Call Extruder 0.16746
  MoveL (T10496) to (109.03, 103.13, 12.7) mm, rotated rx 180 ry 0 rz -180 deg; joints [0, 0, 0, 0, 0, 0]
  Call Extruder 0.05784
  MoveL (T10497) to (109.03, 105.03, 12.7) mm, rotated rx 180 ry 0 rz -180 deg; joints [0, 0, 0, 0, 0, 0]
  Call Extruder 0.08907
  MoveL (T10498) to (111.95, 105.03, 12.7) mm, rotated rx 180 ry 0 rz -180 deg; joints [0, 0, 0, 0, 0, 0]
  Call Extruder 0.05784
  MoveL (T10499) to (111.95, 103.13, 12.7) mm, rotated rx 180 ry 0 rz -180 deg; joints [0, 0, 0, 0, 0, 0]
  Call Extruder 0.00755
  MoveL (T10500) to (112.2, 103.13, 12.7) mm, rotated rx 180 ry 0 rz -180 deg; joints [0, 0, 0, 0, 0, 0]
  Call Extruder 0.05784
  MoveL (T10501) to (112.2, 105.03, 12.7) mm, rotated rx 180 ry 0 rz -180 deg; joints [0, 0, 0, 0, 0, 0]
  Call Extruder 0.08794
  MoveL (T10502) to (115.09, 105.03, 12.7) mm, rotated rx 180 ry 0 rz -180 deg; joints [0, 0, 0, 0, 0, 0]
  Call Extruder 0.05784
  MoveL (T10503) to (115.09, 103.13, 12.7) mm, rotated rx 180 ry 0 rz -180 deg; joints [0, 0, 0, 0, 0, 0]
  Call Extruder 0.20655
  MoveL (T10504) to (121.87, 103.13, 12.7) mm, rotated rx 180 ry 0 rz -180 deg; joints [0, 0, 0, 0, 0, 0]
  Call Extruder 0.16695
  MoveL (T10505) to (121.87, 108.61, 12.7) mm, rotated rx 180 ry 0 rz -180 deg; joints [0, 0, 0, 0, 0, 0]
  Call Extruder 0.05881
  MoveL (T10506) to (119.94, 108.61, 12.7) mm, rotated rx 180 ry 0 rz -180 deg; joints [0, 0, 0, 0, 0, 0]
  Call Extruder 0.09021
  MoveL (T10507) to (119.94, 111.57, 12.7) mm, rotated rx 180 ry 0 rz -180 deg; joints [0, 0, 0, 0, 0, 0]
  Call Extruder 0.05885
  MoveL (T10508) to (121.87, 111.57, 12.7) mm, rotated rx 180 ry 0 rz -180 deg; joints [0, 0, 0, 0, 0, 0]
  Call Extruder 0.02955
  MoveL (T10509) to (121.87, 112.54, 12.7) mm, rotated rx 180 ry 0 rz -180 deg; joints [0, 0, 0, 0, 0, 0]
  Call Extruder 0.05887
  MoveL (T10510) to (119.94, 112.54, 12.7) mm, rotated rx 180 ry 0 rz -180 deg; joints [0, 0, 0, 0, 0, 0]
  Call Extruder 0.08981
  MoveL (T10511) to (119.93, 115.49, 12.7) mm, rotated rx 180 ry 0 rz -180 deg; joints [0, 0, 0, 0, 0, 0]
  Call Extruder 0.05891
  MoveL (T10512) to (121.87, 115.49, 12.7) mm, rotated rx 180 ry 0 rz -180 deg; joints [0, 0, 0, 0, 0, 0]
  Call Extruder 0.19425
  MoveL (T10513) to (121.87, 121.87, 12.7) mm, rotated rx 180 ry 0 rz -180 deg; joints [0, 0, 0, 0, 0, 0]
  Call Extruder 0.57077
  MoveL (T10514) to (103.13, 121.87, 12.7) mm, rotated rx 180 ry 0 rz -180 deg; joints [0, 0, 0, 0, 0, 0]
  Call Extruder 0.57077
  MoveL (T10515) to (103.13, 103.13, 12.7) mm, rotated rx 180 ry 0 rz -180 deg; joints [0, 0, 0, 0, 0, 0]
  Call Extruder 0.01036
  MoveL (T10516) to (103.47, 103.13, 12.7) mm, rotated rx 180 ry 0 rz -180 deg; joints [0, 0, 0, 0, 0, 0]
  Set speed (150.0 mm/s)
  MoveL (T10517) to (102.72, 102.81, 12.7) mm, rotated rx 180 ry 0 rz -180 deg; joints [0, 0, 0, 0, 0, 0]
  Set speed (25.0 mm/s)
  MoveL (T10518) to (102.72, 102.81, 12.7) mm, rotated rx 180 ry 0 rz -180 deg; joints [0, 0, 0, 0, 0, 0]
  Call Extruder 0.00259
  MoveL (T10519) to (102.72, 102.72, 12.7) mm, rotated rx 180 ry 0 rz -180 deg; joints [0, 0, 0, 0, 0, 0]
  Call Extruder 0.20446
  MoveL (T10520) to (109.44, 102.72, 12.7) mm, rotated rx 180 ry 0 rz -180 deg; joints [0, 0, 0, 0, 0, 0]
  Call Extruder 0.05784
  MoveL (T10521) to (109.44, 104.62, 12.7) mm, rotated rx 180 ry 0 rz -180 deg; joints [0, 0, 0, 0, 0, 0]
  Call Extruder 0.06427
  MoveL (T10522) to (111.55, 104.62, 12.7) mm, rotated rx 180 ry 0 rz -180 deg; joints [0, 0, 0, 0, 0, 0]
  Call Extruder 0.05784
  MoveL (T10523) to (111.55, 102.72, 12.7) mm, rotated rx 180 ry 0 rz -180 deg; joints [0, 0, 0, 0, 0, 0]
  Call Extruder 0.03235
  MoveL (T10524) to (112.61, 102.72, 12.7) mm, rotated rx 180 ry 0 rz -180 deg; joints [0, 0, 0, 0, 0, 0]
  Call Extruder 0.05784
  MoveL (T10525) to (112.61, 104.62, 12.7) mm, rotated rx 180 ry 0 rz -180 deg; joints [0, 0, 0, 0, 0, 0]
  Call Extruder 0.06314
  MoveL (T10526) to (114.68, 104.62, 12.7) mm, rotated rx 180 ry 0 rz -180 deg; joints [0, 0, 0, 0, 0, 0]
  Call Extruder 0.05784
  MoveL (T10527) to (114.68, 102.72, 12.7) mm, rotated rx 180 ry 0 rz -180 deg; joints [0, 0, 0, 0, 0, 0]
  Call Extruder 0.23136
  MoveL (T10528) to (122.28, 102.72, 12.7) mm, rotated rx 180 ry 0 rz -180 deg; joints [0, 0, 0, 0, 0, 0]
  Call Extruder 0.19174
  MoveL (T10529) to (122.28, 109.02, 12.7) mm, rotated rx 180 ry 0 rz -180 deg; joints [0, 0, 0, 0, 0, 0]
  Call Extruder 0.05882
  MoveL (T10530) to (120.34, 109.02, 12.7) mm, rotated rx 180 ry 0 rz -180 deg; joints [0, 0, 0, 0, 0, 0]
  Call Extruder 0.06541
  MoveL (T10531) to (120.34, 111.17, 12.7) mm, rotated rx 180 ry 0 rz -180 deg; joints [0, 0, 0, 0, 0, 0]
  Call Extruder 0.05885
  MoveL (T10532) to (122.28, 111.17, 12.7) mm, rotated rx 180 ry 0 rz -180 deg; joints [0, 0, 0, 0, 0, 0]
  Call Extruder 0.05437
  MoveL (T10533) to (122.28, 112.95, 12.7) mm, rotated rx 180 ry 0 rz -180 deg; joints [0, 0, 0, 0, 0, 0]
  Call Extruder 0.05887
  MoveL (T10534) to (120.34, 112.95, 12.7) mm, rotated rx 180 ry 0 rz -180 deg; joints [0, 0, 0, 0, 0, 0]
  Call Extruder 0.06501
  MoveL (T10535) to (120.34, 115.08, 12.7) mm, rotated rx 180 ry 0 rz -180 deg; joints [0, 0, 0, 0, 0, 0]
  Call Extruder 0.0589
  MoveL (T10536) to (122.28, 115.08, 12.7) mm, rotated rx 180 ry 0 rz -180 deg; joints [0, 0, 0, 0, 0, 0]
  Call Extruder 0.21903
  MoveL (T10537) to (122.28, 122.28, 12.7) mm, rotated rx 180 ry 0 rz -180 deg; joints [0, 0, 0, 0, 0, 0]
  Call Extruder 0.59557
  MoveL (T10538) to (102.72, 122.28, 12.7) mm, rotated rx 180 ry 0 rz -180 deg; joints [0, 0, 0, 0, 0, 0]
  Call Extruder 0.59115
  MoveL (T10539) to (102.72, 102.87, 12.7) mm, rotated rx 180 ry 0 rz -180 deg; joints [0, 0, 0, 0, 0, 0]
  Set speed (150.0 mm/s)
  MoveL (T10540) to (102.78, 102.75, 12.7) mm, rotated rx 180 ry 0 rz -180 deg; joints [0, 0, 0, 0, 0, 0]
  Set speed (45.0 mm/s)
  Call Extruder -1.6
  MoveL (T10541) to (102.78, 102.75, 12.7) mm, rotated rx 180 ry 0 rz -180 deg; joints [0, 0, 0, 0, 0, 0]
  Set speed (120.0 mm/s)
  MoveL (T10542) to (102.78, 102.75, 12.7) mm, rotated rx 180 ry 0 rz -180 deg; joints [0, 0, 0, 0, 0, 0]
  Call Extruder -0.05166
  MoveL (T10543) to (102.72, 102.72, 12.7) mm, rotated rx 180 ry 0 rz -180 deg; joints [0, 0, 0, 0, 0, 0]
  Call Extruder -0.32834
  MoveL (T10544) to (103.65, 102.72, 12.7) mm, rotated rx 180 ry 0 rz -180 deg; joints [0, 0, 0, 0, 0, 0]
  Set speed (45.0 mm/s)
  Call Extruder -0.02
  MoveL (T10545) to (103.65, 102.72, 12.7) mm, rotated rx 180 ry 0 rz -180 deg; joints [0, 0, 0, 0, 0, 0]
  Set speed (150.0 mm/s)
  MoveL (T10546) to (103.65, 102.72, 14.7) mm, rotated rx 180 ry 0 rz -180 deg; joints [0, 0, 0, 0, 0, 0]
  MoveL (T10547) to (106.29, 103.84, 14.7) mm, rotated rx 180 ry 0 rz -180 deg; joints [0, 0, 0, 0, 0, 0]
  MoveL (T10548) to (106.29, 103.84, 12.7) mm, rotated rx 180 ry 0 rz -180 deg; joints [0, 0, 0, 0, 0, 0]
  Set speed (40.0 mm/s)
  Call Extruder 2.0
  MoveL (T10549) to (106.29, 103.84, 12.7) mm, rotated rx 180 ry 0 rz -180 deg; joints [0, 0, 0, 0, 0, 0]
  Set speed (26.0 mm/s)
  MoveL (T10550) to (106.29, 103.84, 12.7) mm, rotated rx 180 ry 0 rz -180 deg; joints [0, 0, 0, 0, 0, 0]
  Call Extruder 0.07441
  MoveL (T10551) to (103.84, 103.84, 12.7) mm, rotated rx 180 ry 0 rz -180 deg; joints [0, 0, 0, 0, 0, 0]
  Call Extruder 0.7458
  MoveL (T10552) to (121.16, 121.16, 12.7) mm, rotated rx 180 ry 0 rz -180 deg; joints [0, 0, 0, 0, 0, 0]
  Call Extruder 0.10645
  MoveL (T10553) to (121.16, 117.66, 12.7) mm, rotated rx 180 ry 0 rz -180 deg; joints [0, 0, 0, 0, 0, 0]
  Call Extruder 0.15054
  MoveL (T10554) to (117.66, 121.16, 12.7) mm, rotated rx 180 ry 0 rz -180 deg; joints [0, 0, 0, 0, 0, 0]
  Call Extruder 0.03385
  MoveL (T10555) to (116.55, 121.16, 12.7) mm, rotated rx 180 ry 0 rz -180 deg; joints [0, 0, 0, 0, 0, 0]
  Call Extruder 0.54738
  MoveL (T10556) to (103.84, 108.45, 12.7) mm, rotated rx 180 ry 0 rz -180 deg; joints [0, 0, 0, 0, 0, 0]
  Call Extruder 0.03385
  MoveL (T10557) to (103.84, 107.34, 12.7) mm, rotated rx 180 ry 0 rz -180 deg; joints [0, 0, 0, 0, 0, 0]
  Call Extruder 0.15054
  MoveL (T10558) to (107.34, 103.84, 12.7) mm, rotated rx 180 ry 0 rz -180 deg; joints [0, 0, 0, 0, 0, 0]
  Call Extruder 0.00532
  MoveL (T10559) to (107.51, 103.84, 12.7) mm, rotated rx 180 ry 0 rz -180 deg; joints [0, 0, 0, 0, 0, 0]
  Call Extruder 0.05204
  MoveL (T10560) to (107.51, 105.55, 12.7) mm, rotated rx 180 ry 0 rz -180 deg; joints [0, 0, 0, 0, 0, 0]
  Call Extruder 0.01377
  MoveL (T10561) to (107.83, 105.87, 12.7) mm, rotated rx 180 ry 0 rz -180 deg; joints [0, 0, 0, 0, 0, 0]
  Call Extruder 0.00328
  MoveL (T10562) to (107.94, 105.87, 12.7) mm, rotated rx 180 ry 0 rz -180 deg; joints [0, 0, 0, 0, 0, 0]
  Set speed (45.0 mm/s)
  Call Extruder -1.6
  MoveL (T10563) to (107.94, 105.87, 12.7) mm, rotated rx 180 ry 0 rz -180 deg; joints [0, 0, 0, 0, 0, 0]
  Set speed (120.0 mm/s)
  MoveL (T10564) to (107.94, 105.87, 12.7) mm, rotated rx 180 ry 0 rz -180 deg; joints [0, 0, 0, 0, 0, 0]
  Call Extruder -0.03831
  MoveL (T10565) to (107.83, 105.87, 12.7) mm, rotated rx 180 ry 0 rz -180 deg; joints [0, 0, 0, 0, 0, 0]
  Call Extruder -0.16105
  MoveL (T10566) to (107.51, 105.55, 12.7) mm, rotated rx 180 ry 0 rz -180 deg; joints [0, 0, 0, 0, 0, 0]
  Call Extruder -0.18064
  MoveL (T10567) to (107.51, 105.05, 12.7) mm, rotated rx 180 ry 0 rz -180 deg; joints [0, 0, 0, 0, 0, 0]
  Set speed (45.0 mm/s)
  Call Extruder -0.02
  MoveL (T10568) to (107.51, 105.05, 12.7) mm, rotated rx 180 ry 0 rz -180 deg; joints [0, 0, 0, 0, 0, 0]
  Set speed (150.0 mm/s)
  MoveL (T10569) to (107.51, 105.05, 14.7) mm, rotated rx 180 ry 0 rz -180 deg; joints [0, 0, 0, 0, 0, 0]
  MoveL (T10570) to (107.74, 103.84, 14.7) mm, rotated rx 180 ry 0 rz -180 deg; joints [0, 0, 0, 0, 0, 0]
  MoveL (T10571) to (107.74, 103.84, 12.7) mm, rotated rx 180 ry 0 rz -180 deg; joints [0, 0, 0, 0, 0, 0]
  Set speed (40.0 mm/s)
  Call Extruder 2.0
  MoveL (T10572) to (107.74, 103.84, 12.7) mm, rotated rx 180 ry 0 rz -180 deg; joints [0, 0, 0, 0, 0, 0]
  Set speed (26.0 mm/s)
  MoveL (T10573) to (107.74, 103.84, 12.7) mm, rotated rx 180 ry 0 rz -180 deg; joints [0, 0, 0, 0, 0, 0]
  Call Extruder 0.0285
  MoveL (T10574) to (108.32, 104.42, 12.7) mm, rotated rx 180 ry 0 rz -180 deg; joints [0, 0, 0, 0, 0, 0]
  Call Extruder 0.02289
  MoveL (T10575) to (108.32, 105.08, 12.7) mm, rotated rx 180 ry 0 rz -180 deg; joints [0, 0, 0, 0, 0, 0]
  Call Extruder 0.01949
  MoveL (T10576) to (107.92, 104.69, 12.7) mm, rotated rx 180 ry 0 rz -180 deg; joints [0, 0, 0, 0, 0, 0]
  Call Extruder 0.02289
  MoveL (T10577) to (107.92, 105.34, 12.7) mm, rotated rx 180 ry 0 rz -180 deg; joints [0, 0, 0, 0, 0, 0]
  Call Extruder 0.01503
  MoveL (T10578) to (108.22, 105.65, 12.7) mm, rotated rx 180 ry 0 rz -180 deg; joints [0, 0, 0, 0, 0, 0]
  Set speed (45.0 mm/s)
  Call Extruder -1.6
  MoveL (T10579) to (108.22, 105.65, 12.7) mm, rotated rx 180 ry 0 rz -180 deg; joints [0, 0, 0, 0, 0, 0]
  Set speed (120.0 mm/s)
  MoveL (T10580) to (108.22, 105.65, 12.7) mm, rotated rx 180 ry 0 rz -180 deg; joints [0, 0, 0, 0, 0, 0]
  Call Extruder -0.15379
  MoveL (T10581) to (107.92, 105.34, 12.7) mm, rotated rx 180 ry 0 rz -180 deg; joints [0, 0, 0, 0, 0, 0]
  Call Extruder -0.22621
  MoveL (T10582) to (107.92, 104.71, 12.7) mm, rotated rx 180 ry 0 rz -180 deg; joints [0, 0, 0, 0, 0, 0]
  Set speed (45.0 mm/s)
  Call Extruder -0.02
  MoveL (T10583) to (107.92, 104.71, 12.7) mm, rotated rx 180 ry 0 rz -180 deg; joints [0, 0, 0, 0, 0, 0]
  Set speed (150.0 mm/s)
  MoveL (T10584) to (107.92, 104.71, 14.7) mm, rotated rx 180 ry 0 rz -180 deg; joints [0, 0, 0, 0, 0, 0]
  MoveL (T10585) to (103.84, 109.5, 14.7) mm, rotated rx 180 ry 0 rz -180 deg; joints [0, 0, 0, 0, 0, 0]
  MoveL (T10586) to (103.84, 109.5, 12.7) mm, rotated rx 180 ry 0 rz -180 deg; joints [0, 0, 0, 0, 0, 0]
  Set speed (40.0 mm/s)
  Call Extruder 2.0
  MoveL (T10587) to (103.84, 109.5, 12.7) mm, rotated rx 180 ry 0 rz -180 deg; joints [0, 0, 0, 0, 0, 0]
  Set speed (26.0 mm/s)
  MoveL (T10588) to (103.84, 109.5, 12.7) mm, rotated rx 180 ry 0 rz -180 deg; joints [0, 0, 0, 0, 0, 0]
  Call Extruder 0.07441
  MoveL (T10589) to (103.84, 111.94, 12.7) mm, rotated rx 180 ry 0 rz -180 deg; joints [0, 0, 0, 0, 0, 0]
  Call Extruder 0.26716
  MoveL (T10590) to (110.05, 105.74, 12.7) mm, rotated rx 180 ry 0 rz -180 deg; joints [0, 0, 0, 0, 0, 0]
  Call Extruder 0.00924
  MoveL (T10591) to (110.35, 105.74, 12.7) mm, rotated rx 180 ry 0 rz -180 deg; joints [0, 0, 0, 0, 0, 0]
  Call Extruder 0.38229
  MoveL (T10592) to (119.22, 114.62, 12.7) mm, rotated rx 180 ry 0 rz -180 deg; joints [0, 0, 0, 0, 0, 0]
  Call Extruder 0.01134
  MoveL (T10593) to (119.22, 114.99, 12.7) mm, rotated rx 180 ry 0 rz -180 deg; joints [0, 0, 0, 0, 0, 0]
  Call Extruder 0.26567
  MoveL (T10594) to (113.06, 121.16, 12.7) mm, rotated rx 180 ry 0 rz -180 deg; joints [0, 0, 0, 0, 0, 0]
  Call Extruder 0.03385
  MoveL (T10595) to (111.94, 121.16, 12.7) mm, rotated rx 180 ry 0 rz -180 deg; joints [0, 0, 0, 0, 0, 0]
  Call Extruder 0.34896
  MoveL (T10596) to (103.84, 113.06, 12.7) mm, rotated rx 180 ry 0 rz -180 deg; joints [0, 0, 0, 0, 0, 0]
  Call Extruder 0.10645
  MoveL (T10597) to (103.84, 116.55, 12.7) mm, rotated rx 180 ry 0 rz -180 deg; joints [0, 0, 0, 0, 0, 0]
  Call Extruder 0.46558
  MoveL (T10598) to (114.65, 105.74, 12.7) mm, rotated rx 180 ry 0 rz -180 deg; joints [0, 0, 0, 0, 0, 0]
  Call Extruder 0.00924
  MoveL (T10599) to (114.95, 105.74, 12.7) mm, rotated rx 180 ry 0 rz -180 deg; joints [0, 0, 0, 0, 0, 0]
  Call Extruder 0.18396
  MoveL (T10600) to (119.22, 110.01, 12.7) mm, rotated rx 180 ry 0 rz -180 deg; joints [0, 0, 0, 0, 0, 0]
  Call Extruder 0.01122
  MoveL (T10601) to (119.22, 110.38, 12.7) mm, rotated rx 180 ry 0 rz -180 deg; joints [0, 0, 0, 0, 0, 0]
  Call Extruder 0.46418
  MoveL (T10602) to (108.45, 121.16, 12.7) mm, rotated rx 180 ry 0 rz -180 deg; joints [0, 0, 0, 0, 0, 0]
  Call Extruder 0.03385
  MoveL (T10603) to (107.34, 121.16, 12.7) mm, rotated rx 180 ry 0 rz -180 deg; joints [0, 0, 0, 0, 0, 0]
  Call Extruder 0.15054
  MoveL (T10604) to (103.84, 117.66, 12.7) mm, rotated rx 180 ry 0 rz -180 deg; joints [0, 0, 0, 0, 0, 0]
  Call Extruder 0.10645
  MoveL (T10605) to (103.84, 121.16, 12.7) mm, rotated rx 180 ry 0 rz -180 deg; joints [0, 0, 0, 0, 0, 0]
  Call Extruder 0.7458
  MoveL (T10606) to (121.16, 103.84, 12.7) mm, rotated rx 180 ry 0 rz -180 deg; joints [0, 0, 0, 0, 0, 0]
  Call Extruder 0.09778
  MoveL (T10607) to (121.16, 107.05, 12.7) mm, rotated rx 180 ry 0 rz -180 deg; joints [0, 0, 0, 0, 0, 0]
  Call Extruder 0.00866
  MoveL (T10608) to (120.87, 107.05, 12.7) mm, rotated rx 180 ry 0 rz -180 deg; joints [0, 0, 0, 0, 0, 0]
  Call Extruder 0.13829
  MoveL (T10609) to (117.66, 103.84, 12.7) mm, rotated rx 180 ry 0 rz -180 deg; joints [0, 0, 0, 0, 0, 0]
  Call Extruder 0.02941
  MoveL (T10610) to (116.7, 103.84, 12.7) mm, rotated rx 180 ry 0 rz -180 deg; joints [0, 0, 0, 0, 0, 0]
  Call Extruder 0.045
  MoveL (T10611) to (116.7, 105.32, 12.7) mm, rotated rx 180 ry 0 rz -180 deg; joints [0, 0, 0, 0, 0, 0]
  Set speed (150.0 mm/s)
  MoveL (T10612) to (116.09, 103.66, 12.7) mm, rotated rx 180 ry 0 rz -180 deg; joints [0, 0, 0, 0, 0, 0]
  Set speed (26.0 mm/s)
  MoveL (T10613) to (116.09, 103.66, 12.7) mm, rotated rx 180 ry 0 rz -180 deg; joints [0, 0, 0, 0, 0, 0]
  Call Extruder 0.01001
  MoveL (T10614) to (116.29, 103.86, 12.7) mm, rotated rx 180 ry 0 rz -180 deg; joints [0, 0, 0, 0, 0, 0]
  Call Extruder 0.02527
  MoveL (T10615) to (116.29, 104.55, 12.7) mm, rotated rx 180 ry 0 rz -180 deg; joints [0, 0, 0, 0, 0, 0]
  Call Extruder 0.02525
  MoveL (T10616) to (115.8, 104.06, 12.7) mm, rotated rx 180 ry 0 rz -180 deg; joints [0, 0, 0, 0, 0, 0]
  Call Extruder 0.02527
  MoveL (T10617) to (115.8, 104.75, 12.7) mm, rotated rx 180 ry 0 rz -180 deg; joints [0, 0, 0, 0, 0, 0]
  Call Extruder 0.02525
  MoveL (T10618) to (116.29, 105.24, 12.7) mm, rotated rx 180 ry 0 rz -180 deg; joints [0, 0, 0, 0, 0, 0]
  Call Extruder 0.00537
  MoveL (T10619) to (116.29, 105.38, 12.7) mm, rotated rx 180 ry 0 rz -180 deg; joints [0, 0, 0, 0, 0, 0]
  Call Extruder 0.00419
  MoveL (T10620) to (116.21, 105.47, 12.7) mm, rotated rx 180 ry 0 rz -180 deg; joints [0, 0, 0, 0, 0, 0]
  Call Extruder 0.01395
  MoveL (T10621) to (115.83, 105.47, 12.7) mm, rotated rx 180 ry 0 rz -180 deg; joints [0, 0, 0, 0, 0, 0]
  Call Extruder 0.01079
  MoveL (T10622) to (115.62, 105.26, 12.7) mm, rotated rx 180 ry 0 rz -180 deg; joints [0, 0, 0, 0, 0, 0]
  Set speed (45.0 mm/s)
  Call Extruder -1.6
  MoveL (T10623) to (115.62, 105.26, 12.7) mm, rotated rx 180 ry 0 rz -180 deg; joints [0, 0, 0, 0, 0, 0]
  Set speed (120.0 mm/s)
  MoveL (T10624) to (115.62, 105.26, 12.7) mm, rotated rx 180 ry 0 rz -180 deg; joints [0, 0, 0, 0, 0, 0]
  Call Extruder -0.1051
  MoveL (T10625) to (115.83, 105.47, 12.7) mm, rotated rx 180 ry 0 rz -180 deg; joints [0, 0, 0, 0, 0, 0]
  Call Extruder -0.13599
  MoveL (T10626) to (116.21, 105.47, 12.7) mm, rotated rx 180 ry 0 rz -180 deg; joints [0, 0, 0, 0, 0, 0]
  Call Extruder -0.04087
  MoveL (T10627) to (116.29, 105.38, 12.7) mm, rotated rx 180 ry 0 rz -180 deg; joints [0, 0, 0, 0, 0, 0]
  Call Extruder -0.05236
  MoveL (T10628) to (116.29, 105.24, 12.7) mm, rotated rx 180 ry 0 rz -180 deg; joints [0, 0, 0, 0, 0, 0]
  Call Extruder -0.04569
  MoveL (T10629) to (116.2, 105.15, 12.7) mm, rotated rx 180 ry 0 rz -180 deg; joints [0, 0, 0, 0, 0, 0]
  Set speed (45.0 mm/s)
  Call Extruder -0.02
  MoveL (T10630) to (116.2, 105.15, 12.7) mm, rotated rx 180 ry 0 rz -180 deg; joints [0, 0, 0, 0, 0, 0]
  Set speed (150.0 mm/s)
  MoveL (T10631) to (116.2, 105.15, 14.7) mm, rotated rx 180 ry 0 rz -180 deg; joints [0, 0, 0, 0, 0, 0]
  MoveL (T10632) to (121.34, 107.66, 14.7) mm, rotated rx 180 ry 0 rz -180 deg; joints [0, 0, 0, 0, 0, 0]
  MoveL (T10633) to (121.34, 107.66, 12.7) mm, rotated rx 180 ry 0 rz -180 deg; joints [0, 0, 0, 0, 0, 0]
  Set speed (40.0 mm/s)
  Call Extruder 2.0
  MoveL (T10634) to (121.34, 107.66, 12.7) mm, rotated rx 180 ry 0 rz -180 deg; joints [0, 0, 0, 0, 0, 0]
  Set speed (26.0 mm/s)
  MoveL (T10635) to (121.34, 107.66, 12.7) mm, rotated rx 180 ry 0 rz -180 deg; joints [0, 0, 0, 0, 0, 0]
  Call Extruder 0.00998
  MoveL (T10636) to (121.14, 107.46, 12.7) mm, rotated rx 180 ry 0 rz -180 deg; joints [0, 0, 0, 0, 0, 0]
  Call Extruder 0.02519
  MoveL (T10637) to (120.46, 107.46, 12.7) mm, rotated rx 180 ry 0 rz -180 deg; joints [0, 0, 0, 0, 0, 0]
  Call Extruder 0.02265
  MoveL (T10638) to (120.89, 107.9, 12.7) mm, rotated rx 180 ry 0 rz -180 deg; joints [0, 0, 0, 0, 0, 0]
  Call Extruder 0.02519
  MoveL (T10639) to (120.2, 107.9, 12.7) mm, rotated rx 180 ry 0 rz -180 deg; joints [0, 0, 0, 0, 0, 0]
  Call Extruder 0.02265
  MoveL (T10640) to (119.77, 107.46, 12.7) mm, rotated rx 180 ry 0 rz -180 deg; joints [0, 0, 0, 0, 0, 0]
  Call Extruder 0.00654
  MoveL (T10641) to (119.59, 107.46, 12.7) mm, rotated rx 180 ry 0 rz -180 deg; joints [0, 0, 0, 0, 0, 0]
  Call Extruder 0.00418
  MoveL (T10642) to (119.51, 107.54, 12.7) mm, rotated rx 180 ry 0 rz -180 deg; joints [0, 0, 0, 0, 0, 0]
  Call Extruder 0.01271
  MoveL (T10643) to (119.5, 107.89, 12.7) mm, rotated rx 180 ry 0 rz -180 deg; joints [0, 0, 0, 0, 0, 0]
  Call Extruder 0.00997
  MoveL (T10644) to (119.7, 108.08, 12.7) mm, rotated rx 180 ry 0 rz -180 deg; joints [0, 0, 0, 0, 0, 0]
  Set speed (45.0 mm/s)
  Call Extruder -1.6
  MoveL (T10645) to (119.7, 108.08, 12.7) mm, rotated rx 180 ry 0 rz -180 deg; joints [0, 0, 0, 0, 0, 0]
  Set speed (120.0 mm/s)
  MoveL (T10646) to (119.7, 108.08, 12.7) mm, rotated rx 180 ry 0 rz -180 deg; joints [0, 0, 0, 0, 0, 0]
  Call Extruder -0.09728
  MoveL (T10647) to (119.5, 107.89, 12.7) mm, rotated rx 180 ry 0 rz -180 deg; joints [0, 0, 0, 0, 0, 0]
  Call Extruder -0.12401
  MoveL (T10648) to (119.51, 107.54, 12.7) mm, rotated rx 180 ry 0 rz -180 deg; joints [0, 0, 0, 0, 0, 0]
  Call Extruder -0.04075
  MoveL (T10649) to (119.59, 107.46, 12.7) mm, rotated rx 180 ry 0 rz -180 deg; joints [0, 0, 0, 0, 0, 0]
  Call Extruder -0.06382
  MoveL (T10650) to (119.77, 107.46, 12.7) mm, rotated rx 180 ry 0 rz -180 deg; joints [0, 0, 0, 0, 0, 0]
  Call Extruder -0.05415
  MoveL (T10651) to (119.87, 107.57, 12.7) mm, rotated rx 180 ry 0 rz -180 deg; joints [0, 0, 0, 0, 0, 0]
  Set speed (45.0 mm/s)
  Call Extruder -0.02
  MoveL (T10652) to (119.87, 107.57, 12.7) mm, rotated rx 180 ry 0 rz -180 deg; joints [0, 0, 0, 0, 0, 0]
  Set speed (150.0 mm/s)
  MoveL (T10653) to (119.87, 107.57, 14.7) mm, rotated rx 180 ry 0 rz -180 deg; joints [0, 0, 0, 0, 0, 0]
  MoveL (T10654) to (121.15, 116.79, 14.7) mm, rotated rx 180 ry 0 rz -180 deg; joints [0, 0, 0, 0, 0, 0]
  MoveL (T10655) to (121.15, 116.79, 12.7) mm, rotated rx 180 ry 0 rz -180 deg; joints [0, 0, 0, 0, 0, 0]
  Set speed (40.0 mm/s)
  Call Extruder 2.0
  MoveL (T10656) to (121.15, 116.79, 12.7) mm, rotated rx 180 ry 0 rz -180 deg; joints [0, 0, 0, 0, 0, 0]
  Set speed (26.0 mm/s)
  MoveL (T10657) to (121.15, 116.79, 12.7) mm, rotated rx 180 ry 0 rz -180 deg; joints [0, 0, 0, 0, 0, 0]
  Call Extruder 0.02918
  MoveL (T10658) to (120.56, 116.2, 12.7) mm, rotated rx 180 ry 0 rz -180 deg; joints [0, 0, 0, 0, 0, 0]
  Call Extruder 0.02354
  MoveL (T10659) to (119.89, 116.2, 12.7) mm, rotated rx 180 ry 0 rz -180 deg; joints [0, 0, 0, 0, 0, 0]
  Call Extruder 0.02003
  MoveL (T10660) to (120.3, 116.6, 12.7) mm, rotated rx 180 ry 0 rz -180 deg; joints [0, 0, 0, 0, 0, 0]
  Call Extruder 0.02354
  MoveL (T10661) to (119.63, 116.6, 12.7) mm, rotated rx 180 ry 0 rz -180 deg; joints [0, 0, 0, 0, 0, 0]
  Call Extruder 0.01546
  MoveL (T10662) to (119.32, 116.29, 12.7) mm, rotated rx 180 ry 0 rz -180 deg; joints [0, 0, 0, 0, 0, 0]
  Set speed (45.0 mm/s)
  Call Extruder -1.6
  MoveL (T10663) to (119.32, 116.29, 12.7) mm, rotated rx 180 ry 0 rz -180 deg; joints [0, 0, 0, 0, 0, 0]
  Set speed (120.0 mm/s)
  MoveL (T10664) to (119.32, 116.29, 12.7) mm, rotated rx 180 ry 0 rz -180 deg; joints [0, 0, 0, 0, 0, 0]
  Call Extruder -0.15615
  MoveL (T10665) to (119.63, 116.6, 12.7) mm, rotated rx 180 ry 0 rz -180 deg; joints [0, 0, 0, 0, 0, 0]
  Call Extruder -0.22385
  MoveL (T10666) to (120.26, 116.6, 12.7) mm, rotated rx 180 ry 0 rz -180 deg; joints [0, 0, 0, 0, 0, 0]
  Set speed (45.0 mm/s)
  Call Extruder -0.02
  MoveL (T10667) to (120.26, 116.6, 12.7) mm, rotated rx 180 ry 0 rz -180 deg; joints [0, 0, 0, 0, 0, 0]
  Set speed (150.0 mm/s)
  MoveL (T10668) to (120.26, 116.6, 14.7) mm, rotated rx 180 ry 0 rz -180 deg; joints [0, 0, 0, 0, 0, 0]
  MoveL (T10669) to (104.34, 103.54, 14.7) mm, rotated rx 180 ry 0 rz -180 deg; joints [0, 0, 0, 0, 0, 0]
  MoveL (T10670) to (104.34, 103.54, 12.9) mm, rotated rx 180 ry 0 rz -180 deg; joints [0, 0, 0, 0, 0, 0]
  Set speed (40.0 mm/s)
  Call Extruder 2.0
  MoveL (T10671) to (104.34, 103.54, 12.9) mm, rotated rx 180 ry 0 rz -180 deg; joints [0, 0, 0, 0, 0, 0]
  Set speed (26.3 mm/s)
  MoveL (T10672) to (104.34, 103.54, 12.9) mm, rotated rx 180 ry 0 rz -180 deg; joints [0, 0, 0, 0, 0, 0]
  Call Extruder 0.12704
  MoveL (T10673) to (108.51, 103.54, 12.9) mm, rotated rx 180 ry 0 rz -180 deg; joints [0, 0, 0, 0, 0, 0]
  Call Extruder 0.05785
  MoveL (T10674) to (108.51, 105.44, 12.9) mm, rotated rx 180 ry 0 rz -180 deg; joints [0, 0, 0, 0, 0, 0]
  Call Extruder 0.21676
  MoveL (T10675) to (115.62, 105.44, 12.9) mm, rotated rx 180 ry 0 rz -180 deg; joints [0, 0, 0, 0, 0, 0]
  Call Extruder 0.05785
  MoveL (T10676) to (115.62, 103.54, 12.9) mm, rotated rx 180 ry 0 rz -180 deg; joints [0, 0, 0, 0, 0, 0]
  Call Extruder 0.17785
  MoveL (T10677) to (121.46, 103.54, 12.9) mm, rotated rx 180 ry 0 rz -180 deg; joints [0, 0, 0, 0, 0, 0]
  Call Extruder 0.1385
  MoveL (T10678) to (121.46, 108.09, 12.9) mm, rotated rx 180 ry 0 rz -180 deg; joints [0, 0, 0, 0, 0, 0]
  Call Extruder 0.0588
  MoveL (T10679) to (119.53, 108.09, 12.9) mm, rotated rx 180 ry 0 rz -180 deg; joints [0, 0, 0, 0, 0, 0]
  Call Extruder 0.1151
  MoveL (T10680) to (119.53, 111.86, 12.9) mm, rotated rx 180 ry 0 rz -180 deg; joints [0, 0, 0, 0, 0, 0]
  Call Extruder 0.05885
  MoveL (T10681) to (121.46, 111.86, 12.9) mm, rotated rx 180 ry 0 rz -180 deg; joints [0, 0, 0, 0, 0, 0]
  Call Extruder 0.01167
  MoveL (T10682) to (121.46, 112.25, 12.9) mm, rotated rx 180 ry 0 rz -180 deg; joints [0, 0, 0, 0, 0, 0]
  Call Extruder 0.05885
  MoveL (T10683) to (119.53, 112.25, 12.9) mm, rotated rx 180 ry 0 rz -180 deg; joints [0, 0, 0, 0, 0, 0]
  Call Extruder 0.11468
  MoveL (T10684) to (119.53, 116.01, 12.9) mm, rotated rx 180 ry 0 rz -180 deg; joints [0, 0, 0, 0, 0, 0]
  Call Extruder 0.0589
  MoveL (T10685) to (121.46, 116.01, 12.9) mm, rotated rx 180 ry 0 rz -180 deg; joints [0, 0, 0, 0, 0, 0]
  Call Extruder 0.16601
  MoveL (T10686) to (121.46, 121.46, 12.9) mm, rotated rx 180 ry 0 rz -180 deg; joints [0, 0, 0, 0, 0, 0]
  Call Extruder 0.54596
  MoveL (T10687) to (103.54, 121.46, 12.9) mm, rotated rx 180 ry 0 rz -180 deg; joints [0, 0, 0, 0, 0, 0]
  Call Extruder 0.54596
  MoveL (T10688) to (103.54, 103.54, 12.9) mm, rotated rx 180 ry 0 rz -180 deg; joints [0, 0, 0, 0, 0, 0]
  Call Extruder 0.02254
  MoveL (T10689) to (104.28, 103.54, 12.9) mm, rotated rx 180 ry 0 rz -180 deg; joints [0, 0, 0, 0, 0, 0]
  Set speed (150.0 mm/s)
  MoveL (T10690) to (103.53, 103.13, 12.9) mm, rotated rx 180 ry 0 rz -180 deg; joints [0, 0, 0, 0, 0, 0]
  Set speed (26.3 mm/s)
  MoveL (T10691) to (103.53, 103.13, 12.9) mm, rotated rx 180 ry 0 rz -180 deg; joints [0, 0, 0, 0, 0, 0]
  Call Extruder 0.16404
  MoveL (T10692) to (108.92, 103.13, 12.9) mm, rotated rx 180 ry 0 rz -180 deg; joints [0, 0, 0, 0, 0, 0]
  Call Extruder 0.05785
  MoveL (T10693) to (108.92, 105.03, 12.9) mm, rotated rx 180 ry 0 rz -180 deg; joints [0, 0, 0, 0, 0, 0]
  Call Extruder 0.08906
  MoveL (T10694) to (111.84, 105.03, 12.9) mm, rotated rx 180 ry 0 rz -180 deg; joints [0, 0, 0, 0, 0, 0]
  Call Extruder 0.05785
  MoveL (T10695) to (111.84, 103.13, 12.9) mm, rotated rx 180 ry 0 rz -180 deg; joints [0, 0, 0, 0, 0, 0]
  Call Extruder 0.01484
  MoveL (T10696) to (112.33, 103.13, 12.9) mm, rotated rx 180 ry 0 rz -180 deg; joints [0, 0, 0, 0, 0, 0]
  Call Extruder 0.05785
  MoveL (T10697) to (112.33, 105.03, 12.9) mm, rotated rx 180 ry 0 rz -180 deg; joints [0, 0, 0, 0, 0, 0]
  Call Extruder 0.08799
  MoveL (T10698) to (115.22, 105.03, 12.9) mm, rotated rx 180 ry 0 rz -180 deg; joints [0, 0, 0, 0, 0, 0]
  Call Extruder 0.05785
  MoveL (T10699) to (115.22, 103.13, 12.9) mm, rotated rx 180 ry 0 rz -180 deg; joints [0, 0, 0, 0, 0, 0]
  Call Extruder 0.20266
  MoveL (T10700) to (121.87, 103.13, 12.9) mm, rotated rx 180 ry 0 rz -180 deg; joints [0, 0, 0, 0, 0, 0]
  Call Extruder 0.1633
  MoveL (T10701) to (121.87, 108.49, 12.9) mm, rotated rx 180 ry 0 rz -180 deg; joints [0, 0, 0, 0, 0, 0]
  Call Extruder 0.0588
  MoveL (T10702) to (119.94, 108.49, 12.9) mm, rotated rx 180 ry 0 rz -180 deg; joints [0, 0, 0, 0, 0, 0]
  Call Extruder 0.09029
  MoveL (T10703) to (119.94, 111.46, 12.9) mm, rotated rx 180 ry 0 rz -180 deg; joints [0, 0, 0, 0, 0, 0]
  Call Extruder 0.05884
  MoveL (T10704) to (121.87, 111.46, 12.9) mm, rotated rx 180 ry 0 rz -180 deg; joints [0, 0, 0, 0, 0, 0]
  Call Extruder 0.0365
  MoveL (T10705) to (121.87, 112.66, 12.9) mm, rotated rx 180 ry 0 rz -180 deg; joints [0, 0, 0, 0, 0, 0]
  Call Extruder 0.05886
  MoveL (T10706) to (119.94, 112.65, 12.9) mm, rotated rx 180 ry 0 rz -180 deg; joints [0, 0, 0, 0, 0, 0]
  Call Extruder 0.08988
  MoveL (T10707) to (119.94, 115.6, 12.9) mm, rotated rx 180 ry 0 rz -180 deg; joints [0, 0, 0, 0, 0, 0]
  Call Extruder 0.0589
  MoveL (T10708) to (121.87, 115.61, 12.9) mm, rotated rx 180 ry 0 rz -180 deg; joints [0, 0, 0, 0, 0, 0]
  Call Extruder 0.19079
  MoveL (T10709) to (121.87, 121.87, 12.9) mm, rotated rx 180 ry 0 rz -180 deg; joints [0, 0, 0, 0, 0, 0]
  Call Extruder 0.57077
  MoveL (T10710) to (103.13, 121.87, 12.9) mm, rotated rx 180 ry 0 rz -180 deg; joints [0, 0, 0, 0, 0, 0]
  Call Extruder 0.57077
  MoveL (T10711) to (103.13, 103.13, 12.9) mm, rotated rx 180 ry 0 rz -180 deg; joints [0, 0, 0, 0, 0, 0]
  Call Extruder 0.01036
  MoveL (T10712) to (103.47, 103.13, 12.9) mm, rotated rx 180 ry 0 rz -180 deg; joints [0, 0, 0, 0, 0, 0]
  Set speed (150.0 mm/s)
  MoveL (T10713) to (102.72, 102.81, 12.9) mm, rotated rx 180 ry 0 rz -180 deg; joints [0, 0, 0, 0, 0, 0]
  Set speed (25.0 mm/s)
  MoveL (T10714) to (102.72, 102.81, 12.9) mm, rotated rx 180 ry 0 rz -180 deg; joints [0, 0, 0, 0, 0, 0]
  Call Extruder 0.00259
  MoveL (T10715) to (102.72, 102.72, 12.9) mm, rotated rx 180 ry 0 rz -180 deg; joints [0, 0, 0, 0, 0, 0]
  Call Extruder 0.20103
  MoveL (T10716) to (109.32, 102.72, 12.9) mm, rotated rx 180 ry 0 rz -180 deg; joints [0, 0, 0, 0, 0, 0]
  Call Extruder 0.05785
  MoveL (T10717) to (109.32, 104.62, 12.9) mm, rotated rx 180 ry 0 rz -180 deg; joints [0, 0, 0, 0, 0, 0]
  Call Extruder 0.06426
  MoveL (T10718) to (111.43, 104.62, 12.9) mm, rotated rx 180 ry 0 rz -180 deg; joints [0, 0, 0, 0, 0, 0]
  Call Extruder 0.05785
  MoveL (T10719) to (111.43, 102.72, 12.9) mm, rotated rx 180 ry 0 rz -180 deg; joints [0, 0, 0, 0, 0, 0]
  Call Extruder 0.03963
  MoveL (T10720) to (112.73, 102.72, 12.9) mm, rotated rx 180 ry 0 rz -180 deg; joints [0, 0, 0, 0, 0, 0]
  Call Extruder 0.05785
  MoveL (T10721) to (112.73, 104.62, 12.9) mm, rotated rx 180 ry 0 rz -180 deg; joints [0, 0, 0, 0, 0, 0]
  Call Extruder 0.06319
  MoveL (T10722) to (114.81, 104.62, 12.9) mm, rotated rx 180 ry 0 rz -180 deg; joints [0, 0, 0, 0, 0, 0]
  Call Extruder 0.05785
  MoveL (T10723) to (114.81, 102.72, 12.9) mm, rotated rx 180 ry 0 rz -180 deg; joints [0, 0, 0, 0, 0, 0]
  Call Extruder 0.22746
  MoveL (T10724) to (122.28, 102.72, 12.9) mm, rotated rx 180 ry 0 rz -180 deg; joints [0, 0, 0, 0, 0, 0]
  Call Extruder 0.1881
  MoveL (T10725) to (122.28, 108.9, 12.9) mm, rotated rx 180 ry 0 rz -180 deg; joints [0, 0, 0, 0, 0, 0]
  Call Extruder 0.05881
  MoveL (T10726) to (120.34, 108.9, 12.9) mm, rotated rx 180 ry 0 rz -180 deg; joints [0, 0, 0, 0, 0, 0]
  Call Extruder 0.06549
  MoveL (T10727) to (120.34, 111.05, 12.9) mm, rotated rx 180 ry 0 rz -180 deg; joints [0, 0, 0, 0, 0, 0]
  Call Extruder 0.05884
  MoveL (T10728) to (122.28, 111.05, 12.9) mm, rotated rx 180 ry 0 rz -180 deg; joints [0, 0, 0, 0, 0, 0]
  Call Extruder 0.06132
  MoveL (T10729) to (122.28, 113.06, 12.9) mm, rotated rx 180 ry 0 rz -180 deg; joints [0, 0, 0, 0, 0, 0]
  Call Extruder 0.05886
  MoveL (T10730) to (120.34, 113.06, 12.9) mm, rotated rx 180 ry 0 rz -180 deg; joints [0, 0, 0, 0, 0, 0]
  Call Extruder 0.06508
  MoveL (T10731) to (120.34, 115.2, 12.9) mm, rotated rx 180 ry 0 rz -180 deg; joints [0, 0, 0, 0, 0, 0]
  Call Extruder 0.05889
  MoveL (T10732) to (122.28, 115.2, 12.9) mm, rotated rx 180 ry 0 rz -180 deg; joints [0, 0, 0, 0, 0, 0]
  Call Extruder 0.21558
  MoveL (T10733) to (122.28, 122.28, 12.9) mm, rotated rx 180 ry 0 rz -180 deg; joints [0, 0, 0, 0, 0, 0]
  Call Extruder 0.59557
  MoveL (T10734) to (102.72, 122.28, 12.9) mm, rotated rx 180 ry 0 rz -180 deg; joints [0, 0, 0, 0, 0, 0]
  Call Extruder 0.59115
  MoveL (T10735) to (102.72, 102.87, 12.9) mm, rotated rx 180 ry 0 rz -180 deg; joints [0, 0, 0, 0, 0, 0]
  Set speed (150.0 mm/s)
  MoveL (T10736) to (102.78, 102.75, 12.9) mm, rotated rx 180 ry 0 rz -180 deg; joints [0, 0, 0, 0, 0, 0]
  Set speed (45.0 mm/s)
  Call Extruder -1.6
  MoveL (T10737) to (102.78, 102.75, 12.9) mm, rotated rx 180 ry 0 rz -180 deg; joints [0, 0, 0, 0, 0, 0]
  Set speed (120.0 mm/s)
  MoveL (T10738) to (102.78, 102.75, 12.9) mm, rotated rx 180 ry 0 rz -180 deg; joints [0, 0, 0, 0, 0, 0]
  Call Extruder -0.05166
  MoveL (T10739) to (102.72, 102.72, 12.9) mm, rotated rx 180 ry 0 rz -180 deg; joints [0, 0, 0, 0, 0, 0]
  Call Extruder -0.32834
  MoveL (T10740) to (103.65, 102.72, 12.9) mm, rotated rx 180 ry 0 rz -180 deg; joints [0, 0, 0, 0, 0, 0]
  Set speed (45.0 mm/s)
  Call Extruder -0.02
  MoveL (T10741) to (103.65, 102.72, 12.9) mm, rotated rx 180 ry 0 rz -180 deg; joints [0, 0, 0, 0, 0, 0]
  Set speed (150.0 mm/s)
  MoveL (T10742) to (103.65, 102.72, 14.9) mm, rotated rx 180 ry 0 rz -180 deg; joints [0, 0, 0, 0, 0, 0]
  MoveL (T10743) to (106.29, 103.84, 14.9) mm, rotated rx 180 ry 0 rz -180 deg; joints [0, 0, 0, 0, 0, 0]
  MoveL (T10744) to (106.29, 103.84, 12.9) mm, rotated rx 180 ry 0 rz -180 deg; joints [0, 0, 0, 0, 0, 0]
  Set speed (40.0 mm/s)
  Call Extruder 2.0
  MoveL (T10745) to (106.29, 103.84, 12.9) mm, rotated rx 180 ry 0 rz -180 deg; joints [0, 0, 0, 0, 0, 0]
  Set speed (26.3 mm/s)
  MoveL (T10746) to (106.29, 103.84, 12.9) mm, rotated rx 180 ry 0 rz -180 deg; joints [0, 0, 0, 0, 0, 0]
  Call Extruder 0.07441
  MoveL (T10747) to (103.84, 103.84, 12.9) mm, rotated rx 180 ry 0 rz -180 deg; joints [0, 0, 0, 0, 0, 0]
  Call Extruder 0.7458
  MoveL (T10748) to (121.16, 121.16, 12.9) mm, rotated rx 180 ry 0 rz -180 deg; joints [0, 0, 0, 0, 0, 0]
  Call Extruder 0.10645
  MoveL (T10749) to (121.16, 117.66, 12.9) mm, rotated rx 180 ry 0 rz -180 deg; joints [0, 0, 0, 0, 0, 0]
  Call Extruder 0.15054
  MoveL (T10750) to (117.66, 121.16, 12.9) mm, rotated rx 180 ry 0 rz -180 deg; joints [0, 0, 0, 0, 0, 0]
  Call Extruder 0.03385
  MoveL (T10751) to (116.55, 121.16, 12.9) mm, rotated rx 180 ry 0 rz -180 deg; joints [0, 0, 0, 0, 0, 0]
  Call Extruder 0.54738
  MoveL (T10752) to (103.84, 108.45, 12.9) mm, rotated rx 180 ry 0 rz -180 deg; joints [0, 0, 0, 0, 0, 0]
  Call Extruder 0.03385
  MoveL (T10753) to (103.84, 107.34, 12.9) mm, rotated rx 180 ry 0 rz -180 deg; joints [0, 0, 0, 0, 0, 0]
  Call Extruder 0.15054
  MoveL (T10754) to (107.34, 103.84, 12.9) mm, rotated rx 180 ry 0 rz -180 deg; joints [0, 0, 0, 0, 0, 0]
  Call Extruder 0.00189
  MoveL (T10755) to (107.4, 103.84, 12.9) mm, rotated rx 180 ry 0 rz -180 deg; joints [0, 0, 0, 0, 0, 0]
  Call Extruder 0.05205
  MoveL (T10756) to (107.4, 105.55, 12.9) mm, rotated rx 180 ry 0 rz -180 deg; joints [0, 0, 0, 0, 0, 0]
  Call Extruder 0.01377
  MoveL (T10757) to (107.72, 105.87, 12.9) mm, rotated rx 180 ry 0 rz -180 deg; joints [0, 0, 0, 0, 0, 0]
  Call Extruder 0.0067
  MoveL (T10758) to (107.94, 105.87, 12.9) mm, rotated rx 180 ry 0 rz -180 deg; joints [0, 0, 0, 0, 0, 0]
  Set speed (150.0 mm/s)
  MoveL (T10759) to (108.39, 105.28, 12.9) mm, rotated rx 180 ry 0 rz -180 deg; joints [0, 0, 0, 0, 0, 0]
  Set speed (26.3 mm/s)
  MoveL (T10760) to (108.39, 105.28, 12.9) mm, rotated rx 180 ry 0 rz -180 deg; joints [0, 0, 0, 0, 0, 0]
  Call Extruder 0.00925
  MoveL (T10761) to (108.2, 105.47, 12.9) mm, rotated rx 180 ry 0 rz -180 deg; joints [0, 0, 0, 0, 0, 0]
  Call Extruder 0.01116
  MoveL (T10762) to (107.89, 105.47, 12.9) mm, rotated rx 180 ry 0 rz -180 deg; joints [0, 0, 0, 0, 0, 0]
  Call Extruder 0.00408
  MoveL (T10763) to (107.81, 105.38, 12.9) mm, rotated rx 180 ry 0 rz -180 deg; joints [0, 0, 0, 0, 0, 0]
  Call Extruder 0.00695
  MoveL (T10764) to (107.81, 105.19, 12.9) mm, rotated rx 180 ry 0 rz -180 deg; joints [0, 0, 0, 0, 0, 0]
  Call Extruder 0.01991
  MoveL (T10765) to (108.2, 104.79, 12.9) mm, rotated rx 180 ry 0 rz -180 deg; joints [0, 0, 0, 0, 0, 0]
  Call Extruder 0.02388
  MoveL (T10766) to (108.2, 104.12, 12.9) mm, rotated rx 180 ry 0 rz -180 deg; joints [0, 0, 0, 0, 0, 0]
  Call Extruder 0.01991
  MoveL (T10767) to (107.81, 104.52, 12.9) mm, rotated rx 180 ry 0 rz -180 deg; joints [0, 0, 0, 0, 0, 0]
  Call Extruder 0.02388
  MoveL (T10768) to (107.81, 103.84, 12.9) mm, rotated rx 180 ry 0 rz -180 deg; joints [0, 0, 0, 0, 0, 0]
  Call Extruder 0.00924
  MoveL (T10769) to (107.99, 103.66, 12.9) mm, rotated rx 180 ry 0 rz -180 deg; joints [0, 0, 0, 0, 0, 0]
  Set speed (45.0 mm/s)
  Call Extruder -1.6
  MoveL (T10770) to (107.99, 103.66, 12.9) mm, rotated rx 180 ry 0 rz -180 deg; joints [0, 0, 0, 0, 0, 0]
  Set speed (120.0 mm/s)
  MoveL (T10771) to (107.99, 103.66, 12.9) mm, rotated rx 180 ry 0 rz -180 deg; joints [0, 0, 0, 0, 0, 0]
  Call Extruder -0.09264
  MoveL (T10772) to (107.81, 103.84, 12.9) mm, rotated rx 180 ry 0 rz -180 deg; joints [0, 0, 0, 0, 0, 0]
  Call Extruder -0.23937
  MoveL (T10773) to (107.81, 104.52, 12.9) mm, rotated rx 180 ry 0 rz -180 deg; joints [0, 0, 0, 0, 0, 0]
  Call Extruder -0.04799
  MoveL (T10774) to (107.9, 104.42, 12.9) mm, rotated rx 180 ry 0 rz -180 deg; joints [0, 0, 0, 0, 0, 0]
  Set speed (45.0 mm/s)
  Call Extruder -0.02
  MoveL (T10775) to (107.9, 104.42, 12.9) mm, rotated rx 180 ry 0 rz -180 deg; joints [0, 0, 0, 0, 0, 0]
  Set speed (150.0 mm/s)
  MoveL (T10776) to (107.9, 104.42, 14.9) mm, rotated rx 180 ry 0 rz -180 deg; joints [0, 0, 0, 0, 0, 0]
  MoveL (T10777) to (112.08, 103.34, 14.9) mm, rotated rx 180 ry 0 rz -180 deg; joints [0, 0, 0, 0, 0, 0]
  MoveL (T10778) to (112.08, 103.34, 12.9) mm, rotated rx 180 ry 0 rz -180 deg; joints [0, 0, 0, 0, 0, 0]
  Set speed (40.0 mm/s)
  Call Extruder 2.0
  MoveL (T10779) to (112.08, 103.34, 12.9) mm, rotated rx 180 ry 0 rz -180 deg; joints [0, 0, 0, 0, 0, 0]
  Set speed (26.3 mm/s)
  MoveL (T10780) to (112.08, 103.34, 12.9) mm, rotated rx 180 ry 0 rz -180 deg; joints [0, 0, 0, 0, 0, 0]
  Call Extruder 0.01168
  MoveL (T10781) to (112.08, 105.23, 12.9) mm, rotated rx 180 ry 0 rz -180 deg; joints [0, 0, 0, 0, 0, 0]
  Set speed (45.0 mm/s)
  Call Extruder -1.6
  MoveL (T10782) to (112.08, 105.23, 12.9) mm, rotated rx 180 ry 0 rz -180 deg; joints [0, 0, 0, 0, 0, 0]
  Set speed (120.0 mm/s)
  MoveL (T10783) to (112.08, 105.23, 12.9) mm, rotated rx 180 ry 0 rz -180 deg; joints [0, 0, 0, 0, 0, 0]
  Call Extruder -0.38
  MoveL (T10784) to (112.08, 104.17, 12.9) mm, rotated rx 180 ry 0 rz -180 deg; joints [0, 0, 0, 0, 0, 0]
  Set speed (45.0 mm/s)
  Call Extruder -0.02
  MoveL (T10785) to (112.08, 104.17, 12.9) mm, rotated rx 180 ry 0 rz -180 deg; joints [0, 0, 0, 0, 0, 0]
  Set speed (150.0 mm/s)
  MoveL (T10786) to (112.08, 104.17, 14.9) mm, rotated rx 180 ry 0 rz -180 deg; joints [0, 0, 0, 0, 0, 0]
  MoveL (T10787) to (116.1, 105.65, 14.9) mm, rotated rx 180 ry 0 rz -180 deg; joints [0, 0, 0, 0, 0, 0]
  MoveL (T10788) to (116.1, 105.65, 12.9) mm, rotated rx 180 ry 0 rz -180 deg; joints [0, 0, 0, 0, 0, 0]
  Set speed (40.0 mm/s)
  Call Extruder 2.0
  MoveL (T10789) to (116.1, 105.65, 12.9) mm, rotated rx 180 ry 0 rz -180 deg; joints [0, 0, 0, 0, 0, 0]
  Set speed (26.3 mm/s)
  MoveL (T10790) to (116.1, 105.65, 12.9) mm, rotated rx 180 ry 0 rz -180 deg; joints [0, 0, 0, 0, 0, 0]
  Call Extruder 0.01615
  MoveL (T10791) to (116.42, 105.33, 12.9) mm, rotated rx 180 ry 0 rz -180 deg; joints [0, 0, 0, 0, 0, 0]
  Call Extruder 0.02453
  MoveL (T10792) to (116.42, 104.65, 12.9) mm, rotated rx 180 ry 0 rz -180 deg; joints [0, 0, 0, 0, 0, 0]
  Call Extruder 0.02487
  MoveL (T10793) to (115.93, 105.14, 12.9) mm, rotated rx 180 ry 0 rz -180 deg; joints [0, 0, 0, 0, 0, 0]
  Call Extruder 0.02453
  MoveL (T10794) to (115.93, 104.46, 12.9) mm, rotated rx 180 ry 0 rz -180 deg; joints [0, 0, 0, 0, 0, 0]
  Call Extruder 0.0342
  MoveL (T10795) to (116.6, 103.79, 12.9) mm, rotated rx 180 ry 0 rz -180 deg; joints [0, 0, 0, 0, 0, 0]
  Set speed (150.0 mm/s)
  MoveL (T10796) to (116.82, 105.45, 12.9) mm, rotated rx 180 ry 0 rz -180 deg; joints [0, 0, 0, 0, 0, 0]
  Set speed (26.3 mm/s)
  MoveL (T10797) to (116.82, 105.45, 12.9) mm, rotated rx 180 ry 0 rz -180 deg; joints [0, 0, 0, 0, 0, 0]
  Call Extruder 0.04889
  MoveL (T10798) to (116.82, 103.84, 12.9) mm, rotated rx 180 ry 0 rz -180 deg; joints [0, 0, 0, 0, 0, 0]
  Call Extruder 0.02552
  MoveL (T10799) to (117.66, 103.84, 12.9) mm, rotated rx 180 ry 0 rz -180 deg; joints [0, 0, 0, 0, 0, 0]
  Call Extruder 0.13314
  MoveL (T10800) to (120.75, 106.94, 12.9) mm, rotated rx 180 ry 0 rz -180 deg; joints [0, 0, 0, 0, 0, 0]
  Call Extruder 0.01231
  MoveL (T10801) to (121.16, 106.94, 12.9) mm, rotated rx 180 ry 0 rz -180 deg; joints [0, 0, 0, 0, 0, 0]
  Call Extruder 0.09414
  MoveL (T10802) to (121.16, 103.84, 12.9) mm, rotated rx 180 ry 0 rz -180 deg; joints [0, 0, 0, 0, 0, 0]
  Call Extruder 0.7458
  MoveL (T10803) to (103.84, 121.16, 12.9) mm, rotated rx 180 ry 0 rz -180 deg; joints [0, 0, 0, 0, 0, 0]
  Call Extruder 0.10645
  MoveL (T10804) to (103.84, 117.66, 12.9) mm, rotated rx 180 ry 0 rz -180 deg; joints [0, 0, 0, 0, 0, 0]
  Call Extruder 0.15054
  MoveL (T10805) to (107.34, 121.16, 12.9) mm, rotated rx 180 ry 0 rz -180 deg; joints [0, 0, 0, 0, 0, 0]
  Call Extruder 0.03385
  MoveL (T10806) to (108.45, 121.16, 12.9) mm, rotated rx 180 ry 0 rz -180 deg; joints [0, 0, 0, 0, 0, 0]
  Call Extruder 0.46419
  MoveL (T10807) to (119.22, 110.38, 12.9) mm, rotated rx 180 ry 0 rz -180 deg; joints [0, 0, 0, 0, 0, 0]
  Call Extruder 0.0112
  MoveL (T10808) to (119.22, 110.01, 12.9) mm, rotated rx 180 ry 0 rz -180 deg; joints [0, 0, 0, 0, 0, 0]
  Call Extruder 0.18397
  MoveL (T10809) to (114.95, 105.74, 12.9) mm, rotated rx 180 ry 0 rz -180 deg; joints [0, 0, 0, 0, 0, 0]
  Call Extruder 0.00925
  MoveL (T10810) to (114.65, 105.74, 12.9) mm, rotated rx 180 ry 0 rz -180 deg; joints [0, 0, 0, 0, 0, 0]
  Call Extruder 0.46557
  MoveL (T10811) to (103.84, 116.55, 12.9) mm, rotated rx 180 ry 0 rz -180 deg; joints [0, 0, 0, 0, 0, 0]
  Call Extruder 0.10645
  MoveL (T10812) to (103.84, 113.06, 12.9) mm, rotated rx 180 ry 0 rz -180 deg; joints [0, 0, 0, 0, 0, 0]
  Call Extruder 0.34896
  MoveL (T10813) to (111.94, 121.16, 12.9) mm, rotated rx 180 ry 0 rz -180 deg; joints [0, 0, 0, 0, 0, 0]
  Call Extruder 0.03385
  MoveL (T10814) to (113.06, 121.16, 12.9) mm, rotated rx 180 ry 0 rz -180 deg; joints [0, 0, 0, 0, 0, 0]
  Call Extruder 0.26568
  MoveL (T10815) to (119.22, 114.99, 12.9) mm, rotated rx 180 ry 0 rz -180 deg; joints [0, 0, 0, 0, 0, 0]
  Call Extruder 0.01132
  MoveL (T10816) to (119.22, 114.62, 12.9) mm, rotated rx 180 ry 0 rz -180 deg; joints [0, 0, 0, 0, 0, 0]
  Call Extruder 0.3823
  MoveL (T10817) to (110.35, 105.74, 12.9) mm, rotated rx 180 ry 0 rz -180 deg; joints [0, 0, 0, 0, 0, 0]
  Call Extruder 0.00925
  MoveL (T10818) to (110.05, 105.74, 12.9) mm, rotated rx 180 ry 0 rz -180 deg; joints [0, 0, 0, 0, 0, 0]
  Call Extruder 0.26715
  MoveL (T10819) to (103.84, 111.94, 12.9) mm, rotated rx 180 ry 0 rz -180 deg; joints [0, 0, 0, 0, 0, 0]
  Call Extruder 0.07441
  MoveL (T10820) to (103.84, 109.5, 12.9) mm, rotated rx 180 ry 0 rz -180 deg; joints [0, 0, 0, 0, 0, 0]
  Set speed (45.0 mm/s)
  Call Extruder -1.6
  MoveL (T10821) to (103.84, 109.5, 12.9) mm, rotated rx 180 ry 0 rz -180 deg; joints [0, 0, 0, 0, 0, 0]
  Set speed (120.0 mm/s)
  MoveL (T10822) to (103.84, 109.5, 12.9) mm, rotated rx 180 ry 0 rz -180 deg; joints [0, 0, 0, 0, 0, 0]
  Call Extruder -0.38
  MoveL (T10823) to (103.84, 110.57, 12.9) mm, rotated rx 180 ry 0 rz -180 deg; joints [0, 0, 0, 0, 0, 0]
  Set speed (45.0 mm/s)
  Call Extruder -0.02
  MoveL (T10824) to (103.84, 110.57, 12.9) mm, rotated rx 180 ry 0 rz -180 deg; joints [0, 0, 0, 0, 0, 0]
  Set speed (150.0 mm/s)
  MoveL (T10825) to (103.84, 110.57, 14.9) mm, rotated rx 180 ry 0 rz -180 deg; joints [0, 0, 0, 0, 0, 0]
  MoveL (T10826) to (121.17, 107.16, 14.9) mm, rotated rx 180 ry 0 rz -180 deg; joints [0, 0, 0, 0, 0, 0]
  MoveL (T10827) to (121.17, 107.16, 12.9) mm, rotated rx 180 ry 0 rz -180 deg; joints [0, 0, 0, 0, 0, 0]
  Set speed (40.0 mm/s)
  Call Extruder 2.0
  MoveL (T10828) to (121.17, 107.16, 12.9) mm, rotated rx 180 ry 0 rz -180 deg; joints [0, 0, 0, 0, 0, 0]
  Set speed (26.3 mm/s)
  MoveL (T10829) to (121.17, 107.16, 12.9) mm, rotated rx 180 ry 0 rz -180 deg; joints [0, 0, 0, 0, 0, 0]
  Call Extruder 0.03146
  MoveL (T10830) to (120.55, 107.78, 12.9) mm, rotated rx 180 ry 0 rz -180 deg; joints [0, 0, 0, 0, 0, 0]
  Call Extruder 0.02415
  MoveL (T10831) to (119.87, 107.78, 12.9) mm, rotated rx 180 ry 0 rz -180 deg; joints [0, 0, 0, 0, 0, 0]
  Call Extruder 0.02219
  MoveL (T10832) to (120.31, 107.34, 12.9) mm, rotated rx 180 ry 0 rz -180 deg; joints [0, 0, 0, 0, 0, 0]
  Call Extruder 0.02415
  MoveL (T10833) to (119.64, 107.34, 12.9) mm, rotated rx 180 ry 0 rz -180 deg; joints [0, 0, 0, 0, 0, 0]
  Call Extruder 0.01589
  MoveL (T10834) to (119.32, 107.66, 12.9) mm, rotated rx 180 ry 0 rz -180 deg; joints [0, 0, 0, 0, 0, 0]
  Set speed (45.0 mm/s)
  Call Extruder -1.6
  MoveL (T10835) to (119.32, 107.66, 12.9) mm, rotated rx 180 ry 0 rz -180 deg; joints [0, 0, 0, 0, 0, 0]
  Set speed (120.0 mm/s)
  MoveL (T10836) to (119.32, 107.66, 12.9) mm, rotated rx 180 ry 0 rz -180 deg; joints [0, 0, 0, 0, 0, 0]
  Call Extruder -0.15837
  MoveL (T10837) to (119.64, 107.34, 12.9) mm, rotated rx 180 ry 0 rz -180 deg; joints [0, 0, 0, 0, 0, 0]
  Call Extruder -0.22163
  MoveL (T10838) to (120.26, 107.34, 12.9) mm, rotated rx 180 ry 0 rz -180 deg; joints [0, 0, 0, 0, 0, 0]
  Set speed (45.0 mm/s)
  Call Extruder -0.02
  MoveL (T10839) to (120.26, 107.34, 12.9) mm, rotated rx 180 ry 0 rz -180 deg; joints [0, 0, 0, 0, 0, 0]
  Set speed (150.0 mm/s)
  MoveL (T10840) to (120.26, 107.34, 14.9) mm, rotated rx 180 ry 0 rz -180 deg; joints [0, 0, 0, 0, 0, 0]
  MoveL (T10841) to (121.34, 116.53, 14.9) mm, rotated rx 180 ry 0 rz -180 deg; joints [0, 0, 0, 0, 0, 0]
  MoveL (T10842) to (121.34, 116.53, 12.9) mm, rotated rx 180 ry 0 rz -180 deg; joints [0, 0, 0, 0, 0, 0]
  Set speed (40.0 mm/s)
  Call Extruder 2.0
  MoveL (T10843) to (121.34, 116.53, 12.9) mm, rotated rx 180 ry 0 rz -180 deg; joints [0, 0, 0, 0, 0, 0]
  Set speed (26.3 mm/s)
  MoveL (T10844) to (121.34, 116.53, 12.9) mm, rotated rx 180 ry 0 rz -180 deg; joints [0, 0, 0, 0, 0, 0]
  Call Extruder 0.00965
  MoveL (T10845) to (121.15, 116.72, 12.9) mm, rotated rx 180 ry 0 rz -180 deg; joints [0, 0, 0, 0, 0, 0]
